	(* Valuto se gli assi sono in finestra di prelievo, in questo modo valuto nel ciclo se devo andare fuori ingombro oppure posso partire da dove sono *)
	//IF Mission^.TPick = TPICK_PACK THEN
	(*	(* Valuto la posizione di X *)
		IF (ModuleAx_X^.Ax^.AxRef^.NcToPlc.SetPos >= WorkPickPoint^[Mission^.PPick].Xv - 50) AND (ModuleAx_X^.Ax^.AxRef^.NcToPlc.SetPos <= WorkPickPoint^[Mission^.PPick].Xv + 50) THEN
			AsseXInFinestraDiPrelievoPacco := TRUE;
		ELSE
			AsseXInFinestraDiPrelievoPacco := FALSE;
		END_IF
		
		(* Valuto la rotazione della pinza *)
		IF ModuleAx_J^.Ax^.AxRef^.NcToPlc.SetPos >= Mission^.JPick - 5 AND ModuleAx_J^.Ax^.AxRef^.NcToPlc.SetPos <= Mission^.JPick + 5 THEN
			AsseJInFinestraDiPrelievoPacco := TRUE;
		ELSE
			AsseJInFinestraDiPrelievoPacco := FALSE;
		END_IF
		
		IF Mission^.JPickVO = 0 THEN //Prelievo Verticale
			IF (ModuleAx_Y^.Ax^.AxRef^.NcToPlc.SetPos  >= WorkPickPoint^[Mission^.PPick].Yv - Mission^.YDim/2 - 50) AND (ModuleAx_Y^.Ax^.AxRef^.NcToPlc.SetPos <= WorkPickPoint^[Mission^.PPick].Yv + Mission^.YDim/2 + 50) THEN
				AsseYInFinestraDiPrelievoPacco := TRUE;
			ELSE
				AsseYInFinestraDiPrelievoPacco := FALSE;
			END_IF
		ELSIF Mission^.JPickVO = 1 THEN//Prelievo Orrizontale
			IF (ModuleAx_Y^.Ax^.AxRef^.NcToPlc.SetPos >= WorkPickPoint^[Mission^.PPick].Yh - Mission^.YDim/2 - 50) AND (ModuleAx_Y^.Ax^.AxRef^.NcToPlc.SetPos <= WorkPickPoint^[Mission^.PPick].Yh + Mission^.YDim/2 + 50) THEN
				AsseYInFinestraDiPrelievoPacco := TRUE;
			ELSE
				AsseYInFinestraDiPrelievoPacco := FALSE;
			END_IF
		END_IF
	
	//END_IF
*)

CASE WorkAreaManager^.State OF
	WAMANAGER_NOP,
	
	WAMANAGER_CICLO_RIPOSO_INIT,
		
	WAMANAGER_CICLO_RIPOSO_RUN:
		IF AbilitaAnticipoDinamico THEN
			QuotaAnticipoDinamicaZ_VersoRiposo := 0;
			
			IF TFDirezioneAssePositiva(Posizione_Attuale:=ModuleAX_X^.Ax^.Status.ActPosition,Posizione_Finale:=Mission^.XPick) THEN	// Direzione Positiva 
				TFCalcolaNumeroPostazioneDXSX(PosizioneAttuale:=ModuleAX_X^.Ax^.Status.ActPosition,
												WorkArea:=WorkArea,
												DirezioneAsseX_Positiva:=TRUE,
												NPostazioneDX=>WADX,
												NPostazioneSX=>WASX,
												PostazionePartenza=>WAPARTENZA);
												
				IF WorkArea^[wa].Typology <> TYPOLOGY_EXTERNAL_DEPPREL THEN
					FOR wa := WAPARTENZA TO NumPostazioneDiPareggiatura DO
						AltezzaDiIngombroArea := 0;
						CASE WorkArea^[wa].Typology OF
							
							TYPOLOGY_PALLET:
								CASE Forming^[WorkAreaState^[wa].F].Pallet.Tipologia OF
										
									PALLET_STANDARD:
										IF WorkAreaState^[wa].H > WorkAreaState^[wa].HPL THEN
											AltezzaDiIngombroArea := WorkAreaState^[wa].H;
										ELSE
											AltezzaDiIngombroArea := WorkAreaState^[wa].HPL;
										END_IF
										IF WorkArea^[wa].Z > AltezzaDiIngombroArea THEN
											AltezzaDiIngombroArea := WorkArea^[wa].Z;	
										END_IF
										
									PALLET_ACCOPPIATI:
										IF WorkAreaState^[wa].H > WorkAreaState^[wa].HPL THEN
											AltezzaDiIngombroArea := WorkAreaState^[wa].H;
										ELSE
											AltezzaDiIngombroArea := WorkAreaState^[wa].HPL;
										END_IF
										IF WorkArea^[wa].Z > AltezzaDiIngombroArea THEN
											AltezzaDiIngombroArea := WorkArea^[wa].Z;	
										END_IF	
									
									CASSA_STANDARD:
										IF Forming^[WorkAreaState^[wa].F].Pallet.HMAX > WorkAreaState^[wa].H THEN
											AltezzaDiIngombroArea := Forming^[WorkAreaState^[wa].F].Pallet.HMAX;
										ELSE
											AltezzaDiIngombroArea := WorkAreaState^[wa].H;
										END_IF
										IF WorkArea^[wa].Z > AltezzaDiIngombroArea THEN
											AltezzaDiIngombroArea := WorkArea^[wa].Z;	
										END_IF
										
									CAVALLETTO:
										IF Forming^[WorkAreaState^[wa].F].Pallet.HMAX > WorkAreaState^[wa].H THEN
											AltezzaDiIngombroArea := Forming^[WorkAreaState^[wa].F].Pallet.HMAX;
										ELSE
											AltezzaDiIngombroArea := WorkAreaState^[wa].H;
										END_IF
										IF WorkArea^[wa].Z > AltezzaDiIngombroArea THEN
											AltezzaDiIngombroArea := WorkArea^[wa].Z;	
										END_IF
										
									BUNDLE:
										IF Forming^[WorkAreaState^[wa].F].Pallet.HMAX > WorkAreaState^[wa].H THEN
											AltezzaDiIngombroArea := Forming^[WorkAreaState^[wa].F].Pallet.HMAX;
										ELSE
											AltezzaDiIngombroArea := WorkAreaState^[wa].H;
										END_IF
										IF WorkArea^[wa].Z > AltezzaDiIngombroArea THEN
											AltezzaDiIngombroArea := WorkArea^[wa].Z;	
										END_IF
										
									ELSE
										AltezzaDiIngombroArea := 1700;//Fisso l'altezza ad una quota di default
								END_CASE
											
							TYPOLOGY_LAYER:
								IF WorkAreaState^[wa].H > WorkAreaState^[wa].HPL THEN
									AltezzaDiIngombroArea := WorkAreaState^[wa].H;
								ELSE
									AltezzaDiIngombroArea := WorkAreaState^[wa].HPL;
								END_IF
								IF WorkArea^[wa].Z > AltezzaDiIngombroArea THEN
									AltezzaDiIngombroArea := WorkArea^[wa].Z;	
								END_IF
							
							TYPOLOGY_EXTERNAL_DEPPREL:
								AltezzaDiIngombroArea := AltezzaDiIngombroArea;
								
							ELSE
								AltezzaDiIngombroArea := 1700;//Fisso l'altezza ad una quota di default
						
						END_CASE					
																
						IF QuotaAnticipoDinamicaZ_VersoRiposo <= AltezzaDiIngombroArea + IngombroZ + OffsetSicurezzaAnticipoMovimenti.OffsetSicurezzaAnticipo_Z THEN
							QuotaAnticipoDinamicaZ_VersoRiposo := AltezzaDiIngombroArea + IngombroZ + OffsetSicurezzaAnticipoMovimenti.OffsetSicurezzaAnticipo_Z;
						END_IF
					END_FOR	
					
				END_IF	
				(* Valuto I Pick-Point *)
				CASE TIPOLOGIA_FUNZIONAMENTO_MACCHINA OF
					
					FUNZIONAMENTO_PICKING:
						AltezzaDiIngombroPuntiPrelievo := 0;
															
				ELSE
					FOR P:=1 TO MAXPICKPOINT DO
						AltezzaDiIngombroPuntiPrelievo := 0;
						IF  WorkPickPointDimension^[P].Zdim + WorkPickPointState^[P].Element.Z >= WorkPickPointDimension^[P].Zdim THEN // Se Altezza + Zpacco >= Ingombro Verticale 
							AltezzaDiIngombroPuntiPrelievo := WorkPickPoint^[P].Z + WorkPickPointState^[P].Element.Z;
						END_IF
						IF WorkPickPointDimension^[P].Zdim >= AltezzaDiIngombroPuntiPrelievo THEN //Se Ingombro Verticale >= Dell'ingombro valutato sopra
							AltezzaDiIngombroPuntiPrelievo := WorkPickPointDimension^[P].Zdim;
						END_IF
						//Se non sono nella WA 7, do una quota fittizzia, inferiore all'altezza del ribaltino "reale"
						IF QuotaAnticipoDinamicaZ_VersoRiposo <= AltezzaDiIngombroPuntiPrelievo + TCPParameter.Z + OffsetSicurezzaAnticipoMovimenti.OffsetSicurezzaAnticipo_Z - 300 THEN
							QuotaAnticipoDinamicaZ_VersoRiposo := AltezzaDiIngombroPuntiPrelievo + WorkPickPointState^[P].Element.YDim + TCPParameter.Z + OffsetSicurezzaAnticipoMovimenti.OffsetSicurezzaAnticipo_Z - 300;
						END_IF
					END_FOR			
				END_CASE
				
			ELSE		// Direzione Negativa
				TFCalcolaNumeroPostazioneDXSX(PosizioneAttuale	:= ModuleAX_X^.Ax^.Status.ActPosition,
												WorkArea		:= WorkArea,
												DirezioneAsseX_Positiva:=FALSE,
												NPostazioneDX	=> WADX,
												NPostazioneSX	=> WASX,
												PostazionePartenza=>WAPARTENZA);
						
				FOR wa := WAPARTENZA TO NPOSTAZIONE_DOPODELPUNTODIPREL BY -1 DO
					AltezzaDiIngombroArea := 0;
					IF WorkAreaState^[wa].H > WorkAreaState^[wa].HPL THEN
						AltezzaDiIngombroArea := WorkAreaState^[wa].H;
					ELSE
						AltezzaDiIngombroArea := WorkAreaState^[wa].HPL;
					END_IF
					IF QuotaAnticipoDinamicaZ_VersoRiposo <= AltezzaDiIngombroArea + TCPParameter.Z + OffsetSicurezzaAnticipoMovimenti.OffsetSicurezzaAnticipo_Z THEN
						QuotaAnticipoDinamicaZ_VersoRiposo := AltezzaDiIngombroArea + TCPParameter.Z + OffsetSicurezzaAnticipoMovimenti.OffsetSicurezzaAnticipo_Z;
					END_IF
				END_FOR			
				(* Valuto I Pick-Point *)
				(*FOR P:=1 TO MAXPICKPOINT DO
					AltezzaDiIngombroPuntiPrelievo := 0;
					IF  WorkPickPoint^[P].Zh + WorkPickPointState^[P].ZDim >= WorkPickPointDimension[P].Zdim THEN // Se Altezza orrizzontale Ribaltino + Zpacco >= Ingombro Verticale Ribaltino
						AltezzaDiIngombroPuntiPrelievo := WorkPickPoint^[P].Zh + WorkPickPointState^[P].ZDim;
					END_IF
					IF WorkPickPoint^[P].Zv + WorkPickPointState^[P].ZTilter + WorkPickPointState^[P].YDim >= WorkPickPointDimension[P].Zdim THEN // Se Altezza Vertivale Ribaltino + Quota Fermo + Ypacco >= Ingombro Verticale Ribaltino
						AltezzaDiIngombroPuntiPrelievo := WorkPickPoint^[P].Zv + WorkPickPointState^[P].ZTilter + WorkPickPointState^[P].YDim;
					END_IF
					IF WorkPickPointDimension[P].Zdim >= AltezzaDiIngombroPuntiPrelievo THEN //Se Ingombro Verticale Ribaltino >= Dell'ingombro valutato sopra
						AltezzaDiIngombroPuntiPrelievo := WorkPickPointDimension[P].Zdim;
					END_IF
					IF WAPARTENZA = NPOSTAZIONE_PRIMADELPUNTODIPREL THEN //Se sono nella posizione 7 valuto l'altezza del ribaltino "REALE", con o senza pacco
						IF QuotaAnticipoDinamicaZ_VersoRiposo <= AltezzaDiIngombroPuntiPrelievo + TCPParameter.Z + OffsetSicurezza.Avuoto THEN //Se Quota fuori ingombro <= dell' ingombro del punto di prelievo
							QuotaAnticipoDinamicaZ_VersoRiposo := AltezzaDiIngombroPuntiPrelievo + TCPParameter.Z + OffsetSicurezza.Avuoto;
						END_IF
					ELSE		//Se non sono nella WA 7, do una quota fittizzia, inferiore all'altezza del ribaltino "reale"
						IF QuotaAnticipoDinamicaZ_VersoRiposo <= AltezzaDiIngombroPuntiPrelievo + TCPParameter.Z + OffsetSicurezzaAnticipoMovimenti.OffsetSicurezzaAnticipo_Z - 300 THEN
							QuotaAnticipoDinamicaZ_VersoRiposo := AltezzaDiIngombroPuntiPrelievo + WorkPickPointState^[P].YDim + TCPParameter.Z + OffsetSicurezzaAnticipoMovimenti.OffsetSicurezzaAnticipo_Z - 300;
						END_IF
					END_IF
				END_FOR*)
			END_IF
			IF ModuleAX_Z^.Ax^.Status.ActPosition >= QuotaAnticipoDinamicaZ_VersoRiposo THEN
				QuotaAnticipoDinamicaZ_Raggiunta := TRUE;
			ELSE
				QuotaAnticipoDinamicaZ_Raggiunta := FALSE;
			END_IF
		END_IF
					
										
	WAMANAGER_CICLO_RIPOSO_END,
			
	(*WAMANAGER_CICLO_PALL_INIT,
	
	WAMANAGER_CICLO_PRELIEVO_PALL_RUN:
		(* Calcolo le WA a DX e a SX della mia posizione attuale *)
		WAPARTENZA := Mission^.PPick;
		TFCalcolaNumeroPostazioneDXSX(PosizioneAttuale	:= ModuleAX_X^.Ax^.Status.ActPosition,
										WorkArea		:= WorkArea,
										NPostazioneDX	=> WADX,
										NPostazioneSX	=> WASX);
																
	WAMANAGER_CICLO_PRELIEVO_PALL_END,						
		
	WAMANAGER_CICLO_DEPOSITO_PALL_RUN:
		IF AbilitaAnticipoDinamico THEN
			QuotaAnticipoDinamicaX_DepositoPallet := 0;	
			QuotaAnticipoDinamicaZ_VersoDepPallet := 0;
						
			//IF DirezioneXPositiva_Dep THEN	// Direzione Positiva 
			IF NOT TFDirezioneAssePositiva(Posizione_Attuale:=ModuleAX_X^.Ax^.Status.ActPosition,Posizione_Finale:=Mission^.XPlace) THEN	// Direzione NEGATIVA 
				FOR wa := WAPARTENZA TO Mission^.PPlace BY -1 DO //ordinamento piazzole CRESCENTE CON LA X
					AltezzaDiIngombroArea := 0;
					IF WorkAreaState^[wa].H > WorkAreaState^[wa].HPL THEN
						AltezzaDiIngombroArea := WorkAreaState^[wa].H;
					ELSE
						AltezzaDiIngombroArea := WorkAreaState^[wa].HPL;
					END_IF
					IF QuotaAnticipoDinamicaZ_VersoDepPallet <= AltezzaDiIngombroArea + TCPParameter.Z + OffsetSicurezzaAnticipoMovimenti.OffsetSicurezzaAnticipo_Z THEN
						QuotaAnticipoDinamicaZ_VersoDepPallet := AltezzaDiIngombroArea + TCPParameter.Z + OffsetSicurezzaAnticipoMovimenti.OffsetSicurezzaAnticipo_Z;
					END_IF
				END_FOR		
				(* Valuto I Pick-Point *)
				(*FOR P:=1 TO MAXPICKPOINT DO
					AltezzaDiIngombroPuntiPrelievo := 0;
					IF  WorkPickPoint^[P].Zh + WorkPickPointState^[P].ZDim >= WorkPickPointDimension[P].Zdim THEN // Se Altezza orrizzontale Ribaltino + Zpacco >= Ingombro Verticale Ribaltino
						AltezzaDiIngombroPuntiPrelievo := WorkPickPoint^[P].Zh + WorkPickPointState^[P].ZDim;
					END_IF
					IF WorkPickPoint^[P].Zv + WorkPickPointState^[P].ZTilter + WorkPickPointState^[P].YDim >= WorkPickPointDimension[P].Zdim THEN // Se Altezza Vertivale Ribaltino + Quota Fermo + Ypacco >= Ingombro Verticale Ribaltino
						AltezzaDiIngombroPuntiPrelievo := WorkPickPoint^[P].Zv + WorkPickPointState^[P].ZTilter + WorkPickPointState^[P].YDim;
					END_IF
					IF WorkPickPointDimension[P].Zdim >= AltezzaDiIngombroPuntiPrelievo THEN //Se Ingombro Verticale Ribaltino >= Dell'ingombro valutato sopra
						AltezzaDiIngombroPuntiPrelievo := WorkPickPointDimension[P].Zdim;
					END_IF
					IF WAPARTENZA = NPOSTAZIONE_DOPORIBALTINO THEN //ACR:Se sono nella posizione 7 valuto l'altezza del ribaltino "REALE", con o senza pacco
						IF QuotaAnticipoDinamicaZ_VersoDepPallet <= AltezzaDiIngombroPuntiPrelievo + TCPParameter.Z + OffsetSicurezza.Avuoto THEN //Se Quota fuori ingombro <= dell' ingombro del punto di prelievo
							QuotaAnticipoDinamicaZ_VersoDepPallet := AltezzaDiIngombroPuntiPrelievo + TCPParameter.Z + OffsetSicurezza.Avuoto;
						END_IF
					ELSE		//ACR:Se non sono nella WA 7, do una quota fittizzia, inferiore all'altezza del ribaltino "reale"
						IF QuotaAnticipoDinamicaZ_VersoDepPallet <= AltezzaDiIngombroPuntiPrelievo + TCPParameter.Z + OffsetSicurezzaAnticipoMovimenti.OffsetSicurezzaAnticipo_Z - 300 THEN
							QuotaAnticipoDinamicaZ_VersoDepPallet := AltezzaDiIngombroPuntiPrelievo + WorkPickPointState^[P].YDim + TCPParameter.Z + OffsetSicurezzaAnticipoMovimenti.OffsetSicurezzaAnticipo_Z - 300;
						END_IF
					END_IF
				END_FOR*)
			ELSE		// Direzione POSITIVA
				FOR wa := WAPARTENZA TO Mission^.PPlace DO
					AltezzaDiIngombroArea := 0;
					IF WorkAreaState^[wa].H > WorkAreaState^[wa].HPL THEN
						AltezzaDiIngombroArea := WorkAreaState^[wa].H;
					ELSE
						AltezzaDiIngombroArea := WorkAreaState^[wa].HPL;
					END_IF
					IF QuotaAnticipoDinamicaZ_VersoDepPallet <= AltezzaDiIngombroArea + TCPParameter.Z + OffsetSicurezzaAnticipoMovimenti.OffsetSicurezzaAnticipo_Z THEN
						QuotaAnticipoDinamicaZ_VersoDepPallet := AltezzaDiIngombroArea + TCPParameter.Z + OffsetSicurezzaAnticipoMovimenti.OffsetSicurezzaAnticipo_Z;
					END_IF
				END_FOR			
				(* Valuto I Pick-Point *)
				(*FOR P:=1 TO MAXPICKPOINT DO
					AltezzaDiIngombroPuntiPrelievo := 0;
					IF  WorkPickPoint^[P].Zh + WorkPickPointState^[P].ZDim >= WorkPickPointDimension[P].Zdim THEN // Se Altezza orrizzontale Ribaltino + Zpacco >= Ingombro Verticale Ribaltino
						AltezzaDiIngombroPuntiPrelievo := WorkPickPoint^[P].Zh + WorkPickPointState^[P].ZDim;
					END_IF
					IF WorkPickPoint^[P].Zv + WorkPickPointState^[P].ZTilter + WorkPickPointState^[P].YDim >= WorkPickPointDimension[P].Zdim THEN // Se Altezza Vertivale Ribaltino + Quota Fermo + Ypacco >= Ingombro Verticale Ribaltino
						AltezzaDiIngombroPuntiPrelievo := WorkPickPoint^[P].Zv + WorkPickPointState^[P].ZTilter + WorkPickPointState^[P].YDim;
					END_IF
					IF WorkPickPointDimension[P].Zdim >= AltezzaDiIngombroPuntiPrelievo THEN //Se Ingombro Verticale Ribaltino >= Dell'ingombro valutato sopra
						AltezzaDiIngombroPuntiPrelievo := WorkPickPointDimension[P].Zdim;
					END_IF
					IF WAPARTENZA = NPOSTAZIONE_PRIMADELPUNTODIPREL THEN //Se sono nella posizione 7 valuto l'altezza del ribaltino "REALE", con o senza pacco
						IF QuotaAnticipoDinamicaZ_VersoDepPallet <= AltezzaDiIngombroPuntiPrelievo + TCPParameter.Z + OffsetSicurezza.Avuoto THEN //Se Quota fuori ingombro <= dell' ingombro del punto di prelievo
							QuotaAnticipoDinamicaZ_VersoDepPallet := AltezzaDiIngombroPuntiPrelievo + TCPParameter.Z + OffsetSicurezza.Avuoto;
						END_IF
					ELSE		//Se non sono nella WA 7, do una quota fittizzia, inferiore all'altezza del ribaltino "reale"
						IF QuotaAnticipoDinamicaZ_VersoDepPallet <= AltezzaDiIngombroPuntiPrelievo + TCPParameter.Z + OffsetSicurezzaAnticipoMovimenti.OffsetSicurezzaAnticipo_Z - 300 THEN
							QuotaAnticipoDinamicaZ_VersoDepPallet := AltezzaDiIngombroPuntiPrelievo + WorkPickPointState^[P].YDim + TCPParameter.Z + OffsetSicurezzaAnticipoMovimenti.OffsetSicurezzaAnticipo_Z - 300;
						END_IF
					END_IF
				END_FOR*)
				IF ModuleAX_Z^.Ax^.Status.ActPosition >= QuotaAnticipoDinamicaZ_VersoDepPallet THEN
					QuotaAnticipoDinamicaZ_Raggiunta := TRUE;
				ELSE
					QuotaAnticipoDinamicaZ_Raggiunta := FALSE;
				END_IF	
			END_IF
					
		////////////////// ANTICIPO X ///////////////////////
	(*	IF TFDirezioneAssePositiva(Posizione_Attuale:=ModuleAX_X^.Ax^.Status.ActPosition,Posizione_Finale:=Mission^.XPlace) THEN // Direzione Positiva
			IF Mission^.PPlace <= NPOSTAZIONE_PRIMADELPUNTODIPREL THEN
				IF WorkAreaState^[Mission^.PPlace + 1].P <= 1 THEN
					QuotaAnticipoDinamicaX_DepositoPallet := (Workarea^[Mission^.PPlace + 1].X - Pallet^[Workarea^[Mission^.PPlace + 1].Pallet].X/2 + OffsetSicurezzaAnticipoMovimenti.OffsetSicurezzaAnticipo_X + (IngombroX/2));
				ELSE
					QuotaAnticipoDinamicaX_DepositoPallet := (Workarea^[Mission^.PPlace + 1].X + Pallet^[Workarea^[Mission^.PPlace + 1].Pallet].X/2 + OffsetSicurezzaAnticipoMovimenti.OffsetSicurezzaAnticipo_X + (IngombroX/2));
				END_IF	
			ELSIF Mission^.PPlace > NPOSTAZIONE_DOPORIBALTINO THEN
				IF WorkAreaState^[Mission^.PPlace + 1].P <= 1 THEN
					QuotaAnticipoDinamicaX_DepositoPallet := (Workarea^[Mission^.PPlace + 1].X - Pallet^[Workarea^[Mission^.PPlace + 1].Pallet].X/2 + OffsetSicurezzaAnticipoMovimenti.OffsetSicurezzaAnticipo_X + (IngombroX/2));
				ELSE
					QuotaAnticipoDinamicaX_DepositoPallet := (Workarea^[Mission^.PPlace + 1].X + Pallet^[Workarea^[Mission^.PPlace + 1].Pallet].X/2 + OffsetSicurezzaAnticipoMovimenti.OffsetSicurezzaAnticipo_X + (IngombroX/2));
				END_IF
				IF QuotaAnticipoDinamicaX_DepositoPallet <= Workarea^[NPOSTAZIONE_DOPORIBALTINO].X (*+ 800*) THEN // +800 : In ACR la wa 6 è occupata da falde, questo valore ne indica l'ingombro dal centro verso la wa n° 5
					QuotaAnticipoDinamicaX_DepositoPallet := Workarea^[NPOSTAZIONE_DOPORIBALTINO].X (*+ 800*);
				END_IF
			ELSIF Mission^.PPlace = NPOSTAZIONE_DOPORIBALTINO THEN //postazione 6
				QuotaAnticipoDinamicaX_DepositoPallet := (WorkPickPoint^[Mission^.PPick].Xv + LarghezzaPickPoint/2 + OffsetSicurezzaAnticipoMovimenti.OffsetSicurezzaAnticipo_X + (IngombroX/2));
			END_IF
			IF ModuleAX_X^.Ax^.Status.ActPosition >= QuotaAnticipoDinamicaX_DepositoPallet THEN
				QuotaAnticipoDinamicaX_Raggiunta := TRUE;
			ELSE
				QuotaAnticipoDinamicaX_Raggiunta := FALSE;
			END_IF
		ELSE	//Direzione Negativa
			IF Mission^.PPlace < NPOSTAZIONE_PRIMADELPUNTODIPREL OR Mission^.PPlace >= NPOSTAZIONE_DOPORIBALTINO THEN
				IF WorkAreaState^[Mission^.PPlace - 1].P <= 1 THEN
					QuotaAnticipoDinamicaX_DepositoPallet := (Workarea^[Mission^.PPlace - 1].X + Pallet^[Workarea^[Mission^.PPlace - 1].Pallet].X/2 - OffsetSicurezzaAnticipoMovimenti.OffsetSicurezzaAnticipo_X - (IngombroX/2));
				ELSE
					QuotaAnticipoDinamicaX_DepositoPallet := (Workarea^[Mission^.PPlace - 1].X - Pallet^[Workarea^[Mission^.PPlace - 1].Pallet].X/2 - OffsetSicurezzaAnticipoMovimenti.OffsetSicurezzaAnticipo_X - (IngombroX/2));
				END_IF
			ELSIF Mission^.PPlace = NPOSTAZIONE_PRIMADELPUNTODIPREL THEN
				QuotaAnticipoDinamicaX_DepositoPallet := (WorkPickPoint^[Mission^.PPick].Xv - LarghezzaPickPoint/2 - OffsetSicurezzaAnticipoMovimenti.OffsetSicurezzaAnticipo_X - (IngombroX/2));
			END_IF
			IF ModuleAX_X^.Ax^.Status.ActPosition <= QuotaAnticipoDinamicaX_DepositoPallet THEN
				QuotaAnticipoDinamicaX_Raggiunta := TRUE;
			ELSE
				QuotaAnticipoDinamicaX_Raggiunta := FALSE;
			END_IF
		END_IF*)
		
	END_IF	
				
	WAMANAGER_CICLO_DEPOSITO_PALL_END,
	
	WAMANAGER_CICLO_FALDA_VUOTI_INIT,
	
	WAMANAGER_CICLO_PRELIEVO_FALDA_VUOTI_RUN:
		IF AbilitaAnticipoDinamico THEN
			QuotaAnticipoDinamicaZ_VersoPrelFalda := 0;
				
			//IF DirezioneXPositiva_Prel THEN	// Direzione Positiva 
			IF NOT TFDirezioneAssePositiva(Posizione_Attuale:=ModuleAX_X^.Ax^.Status.ActPosition,Posizione_Finale:=Mission^.XPick) THEN	// Direzione NEGATIVA 
				TFCalcolaNumeroPostazioneDXSX(PosizioneAttuale	:= ModuleAX_X^.Ax^.Status.ActPosition,
												WorkArea		:= WorkArea,
												DirezioneAsseX_Positiva := FALSE,
												NPostazioneDX	=> WADX,
												NPostazioneSX	=> WASX,
												PostazionePartenza=>WAPARTENZA);
				
				FOR wa := WAPARTENZA TO 1 BY -1 DO
					AltezzaDiIngombroArea := 0;
					IF WorkAreaState^[wa].H > WorkAreaState^[wa].HPL THEN
						AltezzaDiIngombroArea := WorkAreaState^[wa].H;
					ELSE
						AltezzaDiIngombroArea := WorkAreaState^[wa].HPL;
					END_IF
					IF QuotaAnticipoDinamicaZ_VersoPrelFalda <= AltezzaDiIngombroArea + TCPParameter.Z + OffsetSicurezzaAnticipoMovimenti.OffsetSicurezzaAnticipo_Z THEN
						QuotaAnticipoDinamicaZ_VersoPrelFalda := AltezzaDiIngombroArea + TCPParameter.Z + OffsetSicurezzaAnticipoMovimenti.OffsetSicurezzaAnticipo_Z;
					END_IF
				END_FOR		
				
				(* Valuto I Pick-Point *)
				(*FOR P:=1 TO MAXPICKPOINT DO
					AltezzaDiIngombroPuntiPrelievo := 0;
					IF  WorkPickPoint^[P].Zh + WorkPickPointState^[P].ZDim >= WorkPickPointDimension[P].Zdim THEN // Se Altezza orrizzontale Ribaltino + Zpacco >= Ingombro Verticale Ribaltino
						AltezzaDiIngombroPuntiPrelievo := WorkPickPoint^[P].Zh + WorkPickPointState^[P].ZDim;
					END_IF
					IF WorkPickPoint^[P].Zv + WorkPickPointState^[P].ZTilter + WorkPickPointState^[P].YDim >= WorkPickPointDimension[P].Zdim THEN // Se Altezza Vertivale Ribaltino + Quota Fermo + Ypacco >= Ingombro Verticale Ribaltino
						AltezzaDiIngombroPuntiPrelievo := WorkPickPoint^[P].Zv + WorkPickPointState^[P].ZTilter + WorkPickPointState^[P].YDim;
					END_IF
					IF WorkPickPointDimension[P].Zdim >= AltezzaDiIngombroPuntiPrelievo THEN //Se Ingombro Verticale Ribaltino >= Dell'ingombro valutato sopra
						AltezzaDiIngombroPuntiPrelievo := WorkPickPointDimension[P].Zdim;
					END_IF
					IF QuotaAnticipoDinamicaZ_VersoPrelFalda <= AltezzaDiIngombroPuntiPrelievo + TCPParameter.Z + OffsetSicurezza.Avuoto THEN //Se Quota fuori ingombro <= dell' ingombro del punto di prelievo
						QuotaAnticipoDinamicaZ_VersoPrelFalda := AltezzaDiIngombroPuntiPrelievo + TCPParameter.Z + OffsetSicurezza.Avuoto;
					END_IF	
				END_FOR*)
				
			ELSE		// Direzione POSITIVA
				FOR wa := WAPARTENZA TO MAXAREA DO
					AltezzaDiIngombroArea := 0;
					IF WorkAreaState^[wa].H > WorkAreaState^[wa].HPL THEN
						AltezzaDiIngombroArea := WorkAreaState^[wa].H;
					ELSE
						AltezzaDiIngombroArea := WorkAreaState^[wa].HPL;
					END_IF
					IF QuotaAnticipoDinamicaZ_VersoPrelFalda <= AltezzaDiIngombroArea + TCPParameter.Z + OffsetSicurezzaAnticipoMovimenti.OffsetSicurezzaAnticipo_Z THEN
						QuotaAnticipoDinamicaZ_VersoPrelFalda := AltezzaDiIngombroArea + TCPParameter.Z + OffsetSicurezzaAnticipoMovimenti.OffsetSicurezzaAnticipo_Z;
					END_IF
				END_FOR			
				(* Valuto I Pick-Point *)
				(*FOR P:=1 TO MAXPICKPOINT DO
					IF Mission^.JPickVO = 0 THEN //Ribaltino Verticale
						IF QuotaAnticipoDinamicaZ_VersoPrelFalda <= WorkPickPoint^[P].Zv + WorkPickPointState^[P].ZTilter + WorkPickPointState^[P].YDim + TCPParameter.Z + OffsetSicurezzaAnticipoMovimenti.OffsetSicurezzaAnticipo_Z THEN
							QuotaAnticipoDinamicaZ_VersoPrelFalda := WorkPickPoint^[P].Zv + WorkPickPointState^[P].ZTilter + WorkPickPointState^[P].YDim + TCPParameter.Z + OffsetSicurezzaAnticipoMovimenti.OffsetSicurezzaAnticipo_Z;
						END_IF
					ELSIF Mission^.JPickVO = 1 THEN	//Ribaltino Orrizontale
						IF QuotaAnticipoDinamicaZ_VersoPrelFalda <= WorkPickPoint^[P].Zh + WorkPickPointState^[P].ZDim + TCPParameter.Z + OffsetSicurezzaAnticipoMovimenti.OffsetSicurezzaAnticipo_Z THEN
							QuotaAnticipoDinamicaZ_VersoPrelFalda := WorkPickPoint^[P].Zh + WorkPickPointState^[P].ZDim + TCPParameter.Z + OffsetSicurezzaAnticipoMovimenti.OffsetSicurezzaAnticipo_Z;
						END_IF
					ELSE
						QuotaAnticipoDinamicaZ_VersoPrelFalda := ALTEZZA_CATASTA_FALDE; // Misura di sicurezza fittizzia
					END_IF
				END_FOR*)
			END_IF
			IF ModuleAX_Z^.Ax^.Status.ActPosition >= QuotaAnticipoDinamicaZ_VersoPrelFalda THEN
				QuotaAnticipoDinamicaZ_Raggiunta := TRUE;
			ELSE
				QuotaAnticipoDinamicaZ_Raggiunta := FALSE;
			END_IF
		END_IF
		
						
	WAMANAGER_CICLO_PRELIEVO_FALDA_VUOTI_END,
		
	WAMANAGER_CICLO_DEPOSITO_FALDA_VUOTI_RUN:
		IF AbilitaAnticipoDinamico THEN
			QuotaAnticipoDinamicaX_VersoDepFalda := 0;
			
			IF TFDirezioneAssePositiva(Posizione_Attuale:=ModuleAX_X^.Ax^.Status.ActPosition,Posizione_Finale:=Mission^.XPlace) THEN
															
				(*IF Mission^.PPlace <= NPOSTAZIONE_PRIMADELPUNTODIPREL THEN
					IF WorkAreaState^[Mission^.PPlace + 1].P <= 1 THEN
						QuotaAnticipoDinamicaX_VersoDepFalda := (Workarea^[Mission^.PPlace + 1].X - Pallet^[Workarea^[Mission^.PPlace + 1].Pallet].X/2 + OffsetSicurezzaAnticipoMovimenti.OffsetSicurezzaAnticipo_X + (IngombroX/2));
					ELSE
						QuotaAnticipoDinamicaX_VersoDepFalda := (Workarea^[Mission^.PPlace + 1].X + Pallet^[Workarea^[Mission^.PPlace + 1].Pallet].X/2 + OffsetSicurezzaAnticipoMovimenti.OffsetSicurezzaAnticipo_X + (IngombroX/2));
					END_IF	
				ELSIF Mission^.PPlace > NPOSTAZIONE_DOPORIBALTINO THEN
					IF WorkAreaState^[Mission^.PPlace + 1].P <= 1 THEN
						QuotaAnticipoDinamicaX_VersoDepFalda := (Workarea^[Mission^.PPlace + 1].X - Pallet^[Workarea^[Mission^.PPlace + 1].Pallet].X/2 + OffsetSicurezzaAnticipoMovimenti.OffsetSicurezzaAnticipo_X + (IngombroX/2));
					ELSE
						QuotaAnticipoDinamicaX_VersoDepFalda := (Workarea^[Mission^.PPlace + 1].X + Pallet^[Workarea^[Mission^.PPlace + 1].Pallet].X/2 + OffsetSicurezzaAnticipoMovimenti.OffsetSicurezzaAnticipo_X + (IngombroX/2));
					END_IF
					IF QuotaAnticipoDinamicaX_VersoDepFalda <= Workarea^[NPOSTAZIONE_DOPORIBALTINO].X + 800 THEN
						QuotaAnticipoDinamicaX_VersoDepFalda := Workarea^[NPOSTAZIONE_DOPORIBALTINO].X + 800;
					END_IF
				ELSIF Mission^.PPlace = NPOSTAZIONE_DOPORIBALTINO THEN //postazione 6
					QuotaAnticipoDinamicaX_VersoDepFalda := (WorkPickPoint^[Mission^.PPick].Xv + LarghezzaPickPoint/2 + OffsetSicurezzaAnticipoMovimenti.OffsetSicurezzaAnticipo_X + (IngombroX/2));
				END_IF
				IF ModuleAX_X^.Ax^.Status.ActPosition >= QuotaAnticipoDinamicaX_VersoDepFalda THEN
					QuotaAnticipoDinamicaX_Raggiunta := TRUE;
				ELSE
					QuotaAnticipoDinamicaX_Raggiunta := FALSE;
				END_IF
			ELSE	//Direzione Negativa
				IF Mission^.PPlace < NPOSTAZIONE_PRIMADELPUNTODIPREL OR Mission^.PPlace >= NPOSTAZIONE_DOPORIBALTINO THEN
					IF WorkAreaState^[Mission^.PPlace - 1].P <= 1 OR WorkArea^[Mission^.PPlace - 1].H + 100 < WorkArea^[Mission^.PPlace].H  THEN
						QuotaAnticipoDinamicaX_VersoDepFalda := (Workarea^[Mission^.PPlace - 1].X + Pallet^[Workarea^[Mission^.PPlace - 1].Pallet].X/2 - OffsetSicurezzaAnticipoMovimenti.OffsetSicurezzaAnticipo_X - (IngombroX/2));
					ELSE
						QuotaAnticipoDinamicaX_VersoDepFalda := (Workarea^[Mission^.PPlace - 1].X - Pallet^[Workarea^[Mission^.PPlace - 1].Pallet].X/2 - OffsetSicurezzaAnticipoMovimenti.OffsetSicurezzaAnticipo_X - (IngombroX/2));
					END_IF
				ELSIF Mission^.PPlace = NPOSTAZIONE_PRIMADELPUNTODIPREL THEN
					QuotaAnticipoDinamicaX_VersoDepFalda := (WorkPickPoint^[Mission^.PPick].Xv - LarghezzaPickPoint/2 - OffsetSicurezzaAnticipoMovimenti.OffsetSicurezzaAnticipo_X - (IngombroX/2));
				END_IF
				IF ModuleAX_X^.Ax^.Status.ActPosition <= QuotaAnticipoDinamicaX_VersoDepFalda THEN
					QuotaAnticipoDinamicaX_Raggiunta := TRUE;
				ELSE
					QuotaAnticipoDinamicaX_Raggiunta := FALSE;
				END_IF*);
			END_IF
		END_IF
											
	WAMANAGER_CICLO_DEPOSITO_FALDA_VUOTI_END,*)
	
	WAMANAGER_CICLO_FALDA_INIT,
	
	WAMANAGER_CICLO_PRELIEVO_FALDA_RUN:
		QuotaAnticipoDinamicaX_Raggiunta := FALSE;
		QuotaAnticipoDinamicaZ_Raggiunta := FALSE;
		QuotaAnticipoDinamicaZ_VersoPrelFalda := 0;
		IF AbilitaAnticipoDinamico THEN
			
			//IF DirezioneXPositiva_Prel THEN	// Direzione Positiva 
			IF NOT TFDirezioneAssePositiva(Posizione_Attuale:=ModuleAX_X^.Ax^.Status.ActPosition,Posizione_Finale:=Mission^.XPlace) THEN	// Direzione NEGATIVA 
				FOR wa := WAPARTENZA TO 1 BY -1 DO
					AltezzaDiIngombroArea := 0;
					IF WorkAreaState^[wa].H > WorkAreaState^[wa].HPL THEN
						AltezzaDiIngombroArea := WorkAreaState^[wa].H;
					ELSE
						AltezzaDiIngombroArea := WorkAreaState^[wa].HPL;
					END_IF
					IF QuotaAnticipoDinamicaZ_VersoPrelFalda <= AltezzaDiIngombroArea + TCPParameter.Z + OffsetSicurezzaAnticipoMovimenti.OffsetSicurezzaAnticipo_Z THEN
						QuotaAnticipoDinamicaZ_VersoPrelFalda := AltezzaDiIngombroArea + TCPParameter.Z + OffsetSicurezzaAnticipoMovimenti.OffsetSicurezzaAnticipo_Z;
					END_IF
				END_FOR		
				
				(* Valuto I Pick-Point *)
				(*FOR P:=1 TO MAXPICKPOINT DO
					AltezzaDiIngombroPuntiPrelievo := 0;
					IF  WorkPickPoint^[P].Zh + WorkPickPointState^[P].ZDim >= WorkPickPointDimension[P].Zdim THEN // Se Altezza orrizzontale Ribaltino + Zpacco >= Ingombro Verticale Ribaltino
						AltezzaDiIngombroPuntiPrelievo := WorkPickPoint^[P].Zh + WorkPickPointState^[P].ZDim;
					END_IF
					IF WorkPickPoint^[P].Zv + WorkPickPointState^[P].ZTilter + WorkPickPointState^[P].YDim >= WorkPickPointDimension[P].Zdim THEN // Se Altezza Vertivale Ribaltino + Quota Fermo + Ypacco >= Ingombro Verticale Ribaltino
						AltezzaDiIngombroPuntiPrelievo := WorkPickPoint^[P].Zv + WorkPickPointState^[P].ZTilter + WorkPickPointState^[P].YDim;
					END_IF
					IF WorkPickPointDimension[P].Zdim >= AltezzaDiIngombroPuntiPrelievo THEN //Se Ingombro Verticale Ribaltino >= Dell'ingombro valutato sopra
						AltezzaDiIngombroPuntiPrelievo := WorkPickPointDimension[P].Zdim;
					END_IF
					IF QuotaAnticipoDinamicaZ_VersoPrelFalda <= AltezzaDiIngombroPuntiPrelievo + TCPParameter.Z + OffsetSicurezza.Avuoto THEN //Se Quota fuori ingombro <= dell' ingombro del punto di prelievo
						QuotaAnticipoDinamicaZ_VersoPrelFalda := AltezzaDiIngombroPuntiPrelievo + TCPParameter.Z + OffsetSicurezza.Avuoto;
					END_IF	
				END_FOR*)
				
			ELSE		// Direzione Negativa
				FOR wa := WAPARTENZA TO MAXAREAPRESENT DO
					AltezzaDiIngombroArea := 0;
					IF WorkAreaState^[wa].H > WorkAreaState^[wa].HPL THEN
						AltezzaDiIngombroArea := WorkAreaState^[wa].H;
					ELSE
						AltezzaDiIngombroArea := WorkAreaState^[wa].HPL;
					END_IF
					IF QuotaAnticipoDinamicaZ_VersoPrelFalda <= AltezzaDiIngombroArea + TCPParameter.Z + OffsetSicurezzaAnticipoMovimenti.OffsetSicurezzaAnticipo_Z THEN
						QuotaAnticipoDinamicaZ_VersoPrelFalda := AltezzaDiIngombroArea + TCPParameter.Z + OffsetSicurezzaAnticipoMovimenti.OffsetSicurezzaAnticipo_Z;
					END_IF
				END_FOR			
				(* Valuto I Pick-Point *)
				(*FOR P:=1 TO MAXPICKPOINT DO
					IF Mission^.JPickVO = 0 THEN //Ribaltino Verticale
						IF QuotaAnticipoDinamicaZ_VersoPrelFalda <= WorkPickPoint^[P].Zv + WorkPickPointState^[P].ZTilter + WorkPickPointState^[P].YDim + TCPParameter.Z + OffsetSicurezzaAnticipoMovimenti.OffsetSicurezzaAnticipo_Z THEN
							QuotaAnticipoDinamicaZ_VersoPrelFalda := WorkPickPoint^[P].Zv + WorkPickPointState^[P].ZTilter + WorkPickPointState^[P].YDim + TCPParameter.Z + OffsetSicurezzaAnticipoMovimenti.OffsetSicurezzaAnticipo_Z;
						END_IF
					ELSIF Mission^.JPickVO = 1 THEN	//Ribaltino Orrizontale
						IF QuotaAnticipoDinamicaZ_VersoPrelFalda <= WorkPickPoint^[P].Zh + WorkPickPointState^[P].ZDim + TCPParameter.Z + OffsetSicurezzaAnticipoMovimenti.OffsetSicurezzaAnticipo_Z THEN
							QuotaAnticipoDinamicaZ_VersoPrelFalda := WorkPickPoint^[P].Zh + WorkPickPointState^[P].ZDim + TCPParameter.Z + OffsetSicurezzaAnticipoMovimenti.OffsetSicurezzaAnticipo_Z;
						END_IF
					ELSE
						QuotaAnticipoDinamicaZ_VersoPrelFalda := ALTEZZA_CATASTA_FALDE; // Misura di sicurezza fittizzia
					END_IF
				END_FOR*)
			END_IF
			IF ModuleAX_Z^.Ax^.Status.ActPosition >= QuotaAnticipoDinamicaZ_VersoPrelFalda THEN
				QuotaAnticipoDinamicaZ_Raggiunta := TRUE;
			ELSE
				QuotaAnticipoDinamicaZ_Raggiunta := FALSE;
			END_IF
		END_IF
		
													
	WAMANAGER_CICLO_PRELIEVO_FALDA_END,
			
	WAMANAGER_CICLO_DEPOSITO_FALDA_RUN:
		IF AbilitaAnticipoDinamico THEN
			QuotaAnticipoDinamicaX_VersoDepFalda := 0;
						
			(*IF TFDirezioneAssePositiva(Posizione_Attuale:=ModuleAX_X^.Ax^.Status.ActPosition,Posizione_Finale:=Mission^.XPlace) THEN
				IF Mission^.PPlace <= NPOSTAZIONE_PRIMADELPUNTODIPREL THEN
					IF WorkAreaState^[Mission^.PPlace + 1].P <= 1 THEN
						QuotaAnticipoDinamicaX_VersoDepFalda := (Workarea^[Mission^.PPlace + 1].X - Pallet^[Workarea^[Mission^.PPlace + 1].Pallet].X/2 + OffsetSicurezzaAnticipoMovimenti.OffsetSicurezzaAnticipo_X + (IngombroX/2));
					ELSE
						QuotaAnticipoDinamicaX_VersoDepFalda := (Workarea^[Mission^.PPlace + 1].X + Pallet^[Workarea^[Mission^.PPlace + 1].Pallet].X/2 + OffsetSicurezzaAnticipoMovimenti.OffsetSicurezzaAnticipo_X + (IngombroX/2));
					END_IF	
				ELSIF Mission^.PPlace > NPOSTAZIONE_DOPORIBALTINO THEN
					IF WorkAreaState^[Mission^.PPlace + 1].P <= 1 THEN
						QuotaAnticipoDinamicaX_VersoDepFalda := (Workarea^[Mission^.PPlace + 1].X - Pallet^[Workarea^[Mission^.PPlace + 1].Pallet].X/2 + OffsetSicurezzaAnticipoMovimenti.OffsetSicurezzaAnticipo_X + (IngombroX/2));
					ELSE
						QuotaAnticipoDinamicaX_VersoDepFalda := (Workarea^[Mission^.PPlace + 1].X + Pallet^[Workarea^[Mission^.PPlace + 1].Pallet].X/2 + OffsetSicurezzaAnticipoMovimenti.OffsetSicurezzaAnticipo_X + (IngombroX/2));
					END_IF
					IF QuotaAnticipoDinamicaX_VersoDepFalda <= Workarea^[NPOSTAZIONE_DOPORIBALTINO].X + 800 THEN
						QuotaAnticipoDinamicaX_VersoDepFalda := Workarea^[NPOSTAZIONE_DOPORIBALTINO].X + 800;
					END_IF
				ELSIF Mission^.PPlace = NPOSTAZIONE_DOPORIBALTINO THEN //postazione 6
					QuotaAnticipoDinamicaX_VersoDepFalda := (WorkPickPoint^[Mission^.PPick].Xv + LarghezzaPickPoint/2 + OffsetSicurezzaAnticipoMovimenti.OffsetSicurezzaAnticipo_X + (IngombroX/2));
				END_IF
				IF ModuleAX_X^.Ax^.Status.ActPosition >= QuotaAnticipoDinamicaX_VersoDepFalda THEN
					QuotaAnticipoDinamicaX_Raggiunta := TRUE;
				ELSE
					QuotaAnticipoDinamicaX_Raggiunta := FALSE;
				END_IF
				TFCalcolaNumeroPostazioneDXSX(PosizioneAttuale	:= ModuleAX_X^.Ax^.Status.ActPosition,
												WorkArea		:= WorkArea,
												DirezioneAsseX_Positiva := TRUE,
												NPostazioneDX	=> WADX,
												NPostazioneSX	=> WASX,
												PostazionePartenza=>WAPARTENZA);
			ELSE	//Direzione Negativa
				IF Mission^.PPlace < NPOSTAZIONE_PRIMADELPUNTODIPREL OR Mission^.PPlace >= NPOSTAZIONE_DOPORIBALTINO THEN
					IF WorkAreaState^[Mission^.PPlace - 1].P <= 1 OR WorkArea^[Mission^.PPlace - 1].H + 100 < WorkArea^[Mission^.PPlace].H  THEN
						QuotaAnticipoDinamicaX_VersoDepFalda := (Workarea^[Mission^.PPlace - 1].X + Pallet^[Workarea^[Mission^.PPlace - 1].Pallet].X/2 - OffsetSicurezzaAnticipoMovimenti.OffsetSicurezzaAnticipo_X - (IngombroX/2));
					ELSE
						QuotaAnticipoDinamicaX_VersoDepFalda := (Workarea^[Mission^.PPlace - 1].X - Pallet^[Workarea^[Mission^.PPlace - 1].Pallet].X/2 - OffsetSicurezzaAnticipoMovimenti.OffsetSicurezzaAnticipo_X - (IngombroX/2));
					END_IF
				ELSIF Mission^.PPlace = NPOSTAZIONE_PRIMADELPUNTODIPREL THEN
					QuotaAnticipoDinamicaX_VersoDepFalda := (WorkPickPoint^[Mission^.PPick].Xv - LarghezzaPickPoint/2 - OffsetSicurezzaAnticipoMovimenti.OffsetSicurezzaAnticipo_X - (IngombroX/2));
				END_IF
				IF ModuleAX_X^.Ax^.Status.ActPosition <= QuotaAnticipoDinamicaX_VersoDepFalda THEN
					QuotaAnticipoDinamicaX_Raggiunta := TRUE;
				ELSE
					QuotaAnticipoDinamicaX_Raggiunta := FALSE;
				END_IF
			END_IF
			TFCalcolaNumeroPostazioneDXSX(PosizioneAttuale	:= ModuleAX_X^.Ax^.Status.ActPosition,
												WorkArea		:= WorkArea,
												DirezioneAsseX_Positiva := FALSE,
												NPostazioneDX	=> WADX,
												NPostazioneSX	=> WASX,
												PostazionePartenza=>WAPARTENZA);
			*)
		END_IF
		WAPARTENZA := Mission^.PPlace;
				
	//WAMANAGER_CICLO_DEPOSITO_FALDA_END,

	(*WAMANAGER_CICLO_PACCO_INIT,
	
	WAMANAGER_CICLO_PRELIEVO_PACCO_RUN:
		IF AbilitaAnticipoDinamico THEN
			QuotaAnticipoDinamicaZ_VersoPrelPacco := 0; 
			//IF DirezioneXPositiva_Prel THEN	// Direzione Positiva 
			IF NOT TFDirezioneAssePositiva(Posizione_Attuale:=ModuleAX_X^.Ax^.Status.ActPosition,Posizione_Finale:=Mission^.XPick) THEN	// Direzione NEGATIVA 
				FOR wa := WAPARTENZA TO NPOSTAZIONE_DOPORIBALTINO BY -1 DO
					AltezzaDiIngombroArea := 0;
					IF WorkAreaState^[wa].H > WorkAreaState^[wa].HPL THEN
						AltezzaDiIngombroArea := WorkAreaState^[wa].H;
					ELSE
						AltezzaDiIngombroArea := WorkAreaState^[wa].HPL;
					END_IF
					IF QuotaAnticipoDinamicaZ_VersoPrelPacco <= AltezzaDiIngombroArea + TCPParameter.Z + OffsetSicurezzaAnticipoMovimenti.OffsetSicurezzaAnticipo_Z THEN
						QuotaAnticipoDinamicaZ_VersoPrelPacco := AltezzaDiIngombroArea + TCPParameter.Z + OffsetSicurezzaAnticipoMovimenti.OffsetSicurezzaAnticipo_Z;
					END_IF
				END_FOR		
				(* Valuto I Pick-Point *)
				(*FOR P:=1 TO MAXPICKPOINT DO
					AltezzaDiIngombroPuntiPrelievo := 0;
					IF  WorkPickPoint^[P].Zh + WorkPickPointState^[P].ZDim >= WorkPickPointDimension[P].Zdim THEN // Se Altezza orrizzontale Ribaltino + Zpacco >= Ingombro Verticale Ribaltino
						AltezzaDiIngombroPuntiPrelievo := WorkPickPoint^[P].Zh + WorkPickPointState^[P].ZDim;
					END_IF
					IF WorkPickPoint^[P].Zv + WorkPickPointState^[P].ZTilter + WorkPickPointState^[P].YDim >= WorkPickPointDimension[P].Zdim THEN // Se Altezza Vertivale Ribaltino + Quota Fermo + Ypacco >= Ingombro Verticale Ribaltino
						AltezzaDiIngombroPuntiPrelievo := WorkPickPoint^[P].Zv + WorkPickPointState^[P].ZTilter + WorkPickPointState^[P].YDim;
					END_IF
					IF WorkPickPointDimension[P].Zdim >= AltezzaDiIngombroPuntiPrelievo THEN //Se Ingombro Verticale Ribaltino >= Dell'ingombro valutato sopra
						AltezzaDiIngombroPuntiPrelievo := WorkPickPointDimension[P].Zdim;
					END_IF
					IF WAPARTENZA = NPOSTAZIONE_DOPORIBALTINO THEN //Se sono nella posizione 7 valuto l'altezza del ribaltino "REALE", con o senza pacco
						IF QuotaAnticipoDinamicaZ_VersoPrelPacco <= AltezzaDiIngombroPuntiPrelievo + TCPParameter.Z + OffsetSicurezza.Avuoto THEN //Se Quota fuori ingombro <= dell' ingombro del punto di prelievo
							QuotaAnticipoDinamicaZ_VersoPrelPacco := AltezzaDiIngombroPuntiPrelievo + TCPParameter.Z + OffsetSicurezza.Avuoto;
						END_IF	
					ELSE
						IF QuotaAnticipoDinamicaZ_VersoPrelPacco <= AltezzaDiIngombroPuntiPrelievo + TCPParameter.Z + OffsetSicurezzaAnticipoMovimenti.OffsetSicurezzaAnticipo_Z - 300 THEN
							QuotaAnticipoDinamicaZ_VersoPrelPacco := AltezzaDiIngombroPuntiPrelievo + WorkPickPointState^[P].YDim + TCPParameter.Z + OffsetSicurezzaAnticipoMovimenti.OffsetSicurezzaAnticipo_Z - 300;
						END_IF
					END_IF
				END_FOR*)
			ELSE		// Direzione POSITIVA
				FOR wa := WAPARTENZA TO NPOSTAZIONE_PRIMADELPUNTODIPREL DO
					AltezzaDiIngombroArea := 0;
					IF WorkAreaState^[wa].H > WorkAreaState^[wa].HPL THEN
						AltezzaDiIngombroArea := WorkAreaState^[wa].H;
					ELSE
						AltezzaDiIngombroArea := WorkAreaState^[wa].HPL;
					END_IF
					IF QuotaAnticipoDinamicaZ_VersoPrelPacco <= AltezzaDiIngombroArea + TCPParameter.Z + OffsetSicurezzaAnticipoMovimenti.OffsetSicurezzaAnticipo_Z THEN
						QuotaAnticipoDinamicaZ_VersoPrelPacco := AltezzaDiIngombroArea + TCPParameter.Z + OffsetSicurezzaAnticipoMovimenti.OffsetSicurezzaAnticipo_Z;
					END_IF
				END_FOR			
								
				(* Valuto I Pick-Point *)
				(*FOR P:=1 TO MAXPICKPOINT DO
					AltezzaDiIngombroPuntiPrelievo := 0;
					IF  WorkPickPoint^[P].Zh + WorkPickPointState^[P].ZDim >= WorkPickPointDimension[P].Zdim THEN // Se Altezza orrizzontale Ribaltino + Zpacco >= Ingombro Verticale Ribaltino
						AltezzaDiIngombroPuntiPrelievo := WorkPickPoint^[P].Zh + WorkPickPointState^[P].ZDim;
					END_IF
					IF WorkPickPoint^[P].Zv + WorkPickPointState^[P].ZTilter + WorkPickPointState^[P].YDim >= WorkPickPointDimension[P].Zdim THEN // Se Altezza Vertivale Ribaltino + Quota Fermo + Ypacco >= Ingombro Verticale Ribaltino
						AltezzaDiIngombroPuntiPrelievo := WorkPickPoint^[P].Zv + WorkPickPointState^[P].ZTilter + WorkPickPointState^[P].YDim;
					END_IF
					IF WorkPickPointDimension[P].Zdim >= AltezzaDiIngombroPuntiPrelievo THEN //Se Ingombro Verticale Ribaltino >= Dell'ingombro valutato sopra
						AltezzaDiIngombroPuntiPrelievo := WorkPickPointDimension[P].Zdim;
					END_IF
					IF WAPARTENZA = NPOSTAZIONE_PRIMADELPUNTODIPREL THEN //Se sono nella posizione 7 valuto l'altezza del ribaltino "REALE", con o senza pacco
						IF QuotaAnticipoDinamicaZ_VersoPrelPacco <= AltezzaDiIngombroPuntiPrelievo + TCPParameter.Z + OffsetSicurezza.Avuoto THEN //Se Quota fuori ingombro <= dell' ingombro del punto di prelievo
							QuotaAnticipoDinamicaZ_VersoPrelPacco := AltezzaDiIngombroPuntiPrelievo + TCPParameter.Z + OffsetSicurezza.Avuoto;
						END_IF
					ELSE		//Se non sono nella WA 7, do una quota fittizzia, inferiore all'altezza del ribaltino "reale"
						IF QuotaAnticipoDinamicaZ_VersoPrelPacco <= AltezzaDiIngombroPuntiPrelievo + TCPParameter.Z + OffsetSicurezzaAnticipoMovimenti.OffsetSicurezzaAnticipo_Z - 300 THEN
							QuotaAnticipoDinamicaZ_VersoPrelPacco := AltezzaDiIngombroPuntiPrelievo + WorkPickPointState^[P].YDim + TCPParameter.Z + OffsetSicurezzaAnticipoMovimenti.OffsetSicurezzaAnticipo_Z - 300;
						END_IF
					END_IF
				END_FOR	*)
			END_IF
				IF ModuleAX_Z^.Ax^.Status.ActPosition >= QuotaAnticipoDinamicaZ_VersoPrelPacco THEN
					QuotaAnticipoDinamicaZ_Raggiunta := TRUE;
				ELSE
					QuotaAnticipoDinamicaZ_Raggiunta := FALSE;
				END_IF
		END_IF
	
				
	WAMANAGER_CICLO_PRELIEVO_PACCO_END,
		
	WAMANAGER_CICLO_DEPOSITO_PACCO_RUN:
		(*IF AbilitaAnticipoDinamico AND Forming^[WorkAreaState^[Mission^.PPlace].F].PackXN[WorkAreaState^[Mission^.PPlace].P].Trajectory <> 2 AND
	    	Forming^[WorkAreaState^[Mission^.PPlace].F].PackXN[WorkAreaState^[Mission^.PPlace].P].Trajectory <> 101 AND
			Forming^[WorkAreaState^[Mission^.PPlace].F].PackXN[WorkAreaState^[Mission^.PPlace].P].Trajectory <> 201 AND
			Forming^[WorkAreaState^[Mission^.PPlace].F].PackXP[WorkAreaState^[Mission^.PPlace].P].Trajectory <> 101 AND
			Forming^[WorkAreaState^[Mission^.PPlace].F].PackXP[WorkAreaState^[Mission^.PPlace].P].Trajectory <> 201 THEN
			QuotaAnticipoDinamicaX_DepositoPacco := 0;
			
			
			//IF DirezioneXPositiva_Dep THEN
			IF NOT TFDirezioneAssePositiva(Posizione_Attuale:=ModuleAX_X^.Ax^.Status.ActPosition,Posizione_Finale:=Mission^.XPlace) THEN
				IF Mission^.PPlace < NPOSTAZIONE_PRIMADELPUNTODIPREL THEN
					IF WorkAreaState^[Mission^.PPlace + 1].P <= 1 THEN
						QuotaAnticipoDinamicaX_DepositoPacco := (Workarea^[Mission^.PPlace + 1].X - Pallet^[Workarea^[Mission^.PPlace + 1].Pallet].X/2 + OffsetSicurezzaAnticipoMovimenti.OffsetSicurezzaAnticipo_X + (IngombroX/2));
					ELSE
						QuotaAnticipoDinamicaX_DepositoPacco := (Workarea^[Mission^.PPlace + 1].X + Pallet^[Workarea^[Mission^.PPlace + 1].Pallet].X/2 + OffsetSicurezzaAnticipoMovimenti.OffsetSicurezzaAnticipo_X + (IngombroX/2));
					END_IF	
				ELSIF Mission^.PPlace > NPOSTAZIONE_DOPORIBALTINO THEN
					IF WorkAreaState^[Mission^.PPlace + 1].P <= 1 THEN
						QuotaAnticipoDinamicaX_DepositoPacco := (Workarea^[Mission^.PPlace + 1].X - Pallet^[Workarea^[Mission^.PPlace + 1].Pallet].X/2 + OffsetSicurezzaAnticipoMovimenti.OffsetSicurezzaAnticipo_X + (IngombroX/2));
					ELSE
						QuotaAnticipoDinamicaX_DepositoPacco := (Workarea^[Mission^.PPlace + 1].X + Pallet^[Workarea^[Mission^.PPlace + 1].Pallet].X/2 + OffsetSicurezzaAnticipoMovimenti.OffsetSicurezzaAnticipo_X + (IngombroX/2));
					END_IF
					//IF QuotaAnticipoDinamicaX_DepositoPacco <= Workarea^[NPOSTAZIONE_DOPORIBALTINO].X + 800 + (IngombroX/2) + OffsetSicurezzaAnticipoMovimenti.OffsetSicurezzaAnticipo_X THEN
					//	QuotaAnticipoDinamicaX_DepositoPacco := Workarea^[NPOSTAZIONE_DOPORIBALTINO].X + 800 + (IngombroX/2) + OffsetSicurezzaAnticipoMovimenti.OffsetSicurezzaAnticipo_X;
					//END_IF
				ELSIF Mission^.PPlace = NPOSTAZIONE_DOPORIBALTINO OR Mission^.PPlace = NPOSTAZIONE_PRIMADELPUNTODIPREL THEN //postazione 5,6
					QuotaAnticipoDinamicaX_DepositoPacco := (WorkPickPoint^[Mission^.PPick].Xv + LarghezzaPickPoint/2 + OffsetSicurezzaAnticipoMovimenti.OffsetSicurezzaAnticipo_X + (IngombroX/2));
				END_IF
				IF ModuleAX_X^.Ax^.Status.ActPosition <= QuotaAnticipoDinamicaX_DepositoPacco THEN
					QuotaAnticipoDinamicaX_Raggiunta := TRUE;
				ELSE
					QuotaAnticipoDinamicaX_Raggiunta := FALSE;
				END_IF
				TFCalcolaNumeroPostazioneDXSX(PosizioneAttuale	:= ModuleAX_X^.Ax^.Status.ActPosition,
												WorkArea		:= WorkArea,
												DirezioneAsseX_Positiva := FALSE,
												NPostazioneDX	=> WADX,
												NPostazioneSX	=> WASX,
												PostazionePartenza=>WAPARTENZA);
			ELSE	//Direzione POSITIVA
				IF Mission^.PPlace < NPOSTAZIONE_PRIMADELPUNTODIPREL OR Mission^.PPlace > NPOSTAZIONE_DOPORIBALTINO THEN
					IF WorkAreaState^[Mission^.PPlace - 1].P <= 1 OR WorkArea^[Mission^.PPlace - 1].H + 100 < WorkArea^[Mission^.PPlace].H  THEN
						QuotaAnticipoDinamicaX_DepositoPacco := (Workarea^[Mission^.PPlace - 1].X + Pallet^[Workarea^[Mission^.PPlace - 1].Pallet].X/2 - OffsetSicurezzaAnticipoMovimenti.OffsetSicurezzaAnticipo_X - (IngombroX/2));
					ELSE
						QuotaAnticipoDinamicaX_DepositoPacco := (Workarea^[Mission^.PPlace - 1].X - Pallet^[Workarea^[Mission^.PPlace - 1].Pallet].X/2 - OffsetSicurezzaAnticipoMovimenti.OffsetSicurezzaAnticipo_X - (IngombroX/2));
					END_IF
				ELSIF Mission^.PPlace = NPOSTAZIONE_PRIMADELPUNTODIPREL OR  Mission^.PPlace = NPOSTAZIONE_DOPORIBALTINO THEN
					QuotaAnticipoDinamicaX_DepositoPacco := (WorkPickPoint^[Mission^.PPick].Xv - LarghezzaPickPoint/2 - OffsetSicurezzaAnticipoMovimenti.OffsetSicurezzaAnticipo_X - (IngombroX/2));
				END_IF
				IF ModuleAX_X^.Ax^.Status.ActPosition >= QuotaAnticipoDinamicaX_DepositoPacco THEN
					QuotaAnticipoDinamicaX_Raggiunta := TRUE;
				ELSE
					QuotaAnticipoDinamicaX_Raggiunta := FALSE;
				END_IF
				TFCalcolaNumeroPostazioneDXSX(PosizioneAttuale	:= ModuleAX_X^.Ax^.Status.ActPosition,
												WorkArea		:= WorkArea,
												DirezioneAsseX_Positiva := TRUE,
												NPostazioneDX	=> WADX,
												NPostazioneSX	=> WASX,
												PostazionePartenza=>WAPARTENZA);
			END_IF
		END_IF*)
		
		WAPARTENZA := Mission^.PPlace;
				
	//WAMANAGER_CICLO_DEPOSITO_PACCO_END;
	*)
END_CASE

END_FUNCTION_BLOCK

// ---- POUs/TFPalletizerDataTF/TFValutaAssiInFinestraDiPassMode.TcPOU
FUNCTION_BLOCK TFValutaAssiInFinestraDiPassMode
VAR_INPUT
	ModuleAX_X : POINTER TO TFModulePalletizer_Ax;
	ModuleAX_Y : POINTER TO TFModulePalletizer_Ax;
	ModuleAX_Z : POINTER TO TFModulePalletizer_Ax;
	ModuleAX_J : POINTER TO TFModulePalletizer_AxJ_Lastre;
	Traiettoria : POINTER TO TFTraiettoria;
	WorkAreaManager : POINTER TO TFWorkAreaManager;
END_VAR
VAR
	Direzione_X_Positiva : BOOL;
	Direzione_Y_Positiva : BOOL;
	Direzione_Z_Positiva : BOOL;
	Direzione_J_Positiva : BOOL;
	Direzione_K_Positiva : bool;
	AsseXInMoto: BOOL;
	AsseYInMoto: BOOL;
	AsseZInMoto: BOOL;
	AsseJInMoto: BOOL;
	//AsseKInMoto: BOOL;
	OffsetPassModeY_Appoggio: REAL;
END_VAR

(* Azzero le variabili *)
Asse_X_InFinestraDiPassMode := FALSE;
Asse_Y_InFinestraDiPassMode := FALSE;
Asse_Z_InFinestraDiPassMode := FALSE;
Asse_J_InFinestraDiPassMode := FALSE;

(* Valuto la direzione degli assi *)
Direzione_X_Positiva := TFDirezioneAssePositiva(Posizione_Attuale:=ModuleAX_X^.Ax^.Status.ActPosition,Posizione_Finale:=ProgrammaToModule_X.Quota_Destinazione);
Direzione_Y_Positiva := TFDirezioneAssePositiva(Posizione_Attuale:=ModuleAX_Y^.Ax^.Status.ActPosition,Posizione_Finale:=ProgrammaToModule_Y.Quota_Destinazione);
Direzione_Z_Positiva := TFDirezioneAssePositiva(Posizione_Attuale:=ModuleAX_Z^.Ax^.Status.ActPosition,Posizione_Finale:=ProgrammaToModule_Z.Quota_Destinazione);
Direzione_J_Positiva := TFDirezioneAssePositiva(Posizione_Attuale:=ModuleAX_J^.Ax^.Status.ActPosition,Posizione_Finale:=ProgrammaToModule_J.Quota_Destinazione);
(* Valuto se gli assi si stanno muovendo *)
AsseXInMoto:=ModuleAX_X^.Ax^.AxRef^.Status.Moving;
AsseYInMoto:=ModuleAX_Y^.Ax^.AxRef^.Status.Moving;
AsseZInMoto:=ModuleAX_Z^.Ax^.AxRef^.Status.Moving;
AsseJInMoto:=ModuleAX_J^.Ax^.AxRef^.Status.Moving;

IF Traiettoria^.PassModeGlobalEnable AND AbilitazionePassModeGlobale THEN (* Abilitazione Globale del PassMode*)
	
//	CASE WorkAreaManager^.State OF
		
//		WAMANAGER_CICLO_RIPOSO_RUN: 
			(* Abilito tutti i pasmode*)
			Traiettoria^.PassModePoint_X_Enable[1] := TRUE; 
			Traiettoria^.PassModePoint_Y_Enable[1] := TRUE; 
			Traiettoria^.PassModePoint_Z_Enable[1] := TRUE;
			Traiettoria^.PassModePoint_J_Enable[1] := TRUE;
			Traiettoria^.PassModePoint_K_Enable[1] := TRUE;
			(* Valuta il Pass Mode Per L'asse X *)
			IF Traiettoria^.PassModePoint_X_Enable[1] THEN
				IF AsseXInMoto THEN
					IF Direzione_X_Positiva THEN	//Se l'asse si sta muovendo in direzione POSITIVA
						IF ModuleAX_X^.Ax^.Status.ActPosition >= (ProgrammaToModule_X.Quota_Destinazione - OffsetPassMode.X) THEN
							Asse_X_InFinestraDiPassMode := TRUE;	
						END_IF
					ELSE							//Se l'asse si sta muovendo in direzione NEGATIVA
						IF ModuleAX_X^.Ax^.Status.ActPosition <= (ProgrammaToModule_X.Quota_Destinazione + OffsetPassMode.X) THEN
							Asse_X_InFinestraDiPassMode := TRUE;	
						END_IF
					END_IF
				END_IF
			END_IF
				
			(* Valuta il Pass Mode Per L'asse Y *)
			IF Traiettoria^.PassModePoint_Y_Enable[1] THEN
				IF Pinza_InIngombroColonne_Attuale THEN
					OffsetPassModeY_Appoggio := 80;
				ELSE
					OffsetPassModeY_Appoggio := OffsetPassMode.Y;
				END_IF
				IF AsseYInMoto THEN
					IF Direzione_Y_Positiva THEN	//Se l'asse si sta muovendo in direzione POSITIVA
						IF ModuleAX_Y^.Ax^.Status.ActPosition >= (ProgrammaToModule_Y.Quota_Destinazione - OffsetPassModeY_Appoggio) THEN
							Asse_Y_InFinestraDiPassMode := TRUE;	
						END_IF
					ELSE							//Se l'asse si sta muovendo in direzione NEGATIVA
						IF ModuleAX_Y^.Ax^.Status.ActPosition <= (ProgrammaToModule_Y.Quota_Destinazione + OffsetPassModeY_Appoggio) THEN
							Asse_Y_InFinestraDiPassMode := TRUE;	
						END_IF
					END_IF
				END_IF
			END_IF
			
			(* Valuta il Pass Mode Per L'asse Z *)
			IF Traiettoria^.PassModePoint_Z_Enable[1] THEN
				IF AsseZInMoto THEN
					IF Direzione_Z_Positiva THEN	//Se l'asse si sta muovendo in direzione POSITIVA
						IF ModuleAX_Z^.Ax^.Status.ActPosition >= (ProgrammaToModule_Z.Quota_Destinazione - OffsetPassMode.Z) THEN
							Asse_Z_InFinestraDiPassMode := TRUE;	
						END_IF
					ELSE							//Se l'asse si sta muovendo in direzione NEGATIVA
						IF ModuleAX_Z^.Ax^.Status.ActPosition <= (ProgrammaToModule_Z.Quota_Destinazione + OffsetPassMode.Z) THEN
							Asse_Z_InFinestraDiPassMode := TRUE;	
						END_IF
					END_IF
				END_IF
			END_IF
			
			(* Valuta il Pass Mode Per L'asse J *)
			IF Traiettoria^.PassModePoint_J_Enable[1] THEN
				IF AsseJInMoto THEN
					IF Direzione_J_Positiva THEN	//Se l'asse si sta muovendo in direzione POSITIVA
						IF ModuleAX_J^.Ax^.Status.ActPosition >= (ProgrammaToModule_J.Quota_Destinazione - OffsetPassMode.J) THEN
							Asse_J_InFinestraDiPassMode := TRUE;	
						END_IF
					ELSE							//Se l'asse si sta muovendo in direzione NEGATIVA
						IF ModuleAX_J^.Ax^.Status.ActPosition <= (ProgrammaToModule_J.Quota_Destinazione + OffsetPassMode.J) THEN
							Asse_J_InFinestraDiPassMode := TRUE;	
						END_IF
					END_IF
				END_IF
			END_IF
		(*
		WAMANAGER_CICLO_PRELIEVO_PALL_RUN: 
			(* Abilito tutti i pasmode*)
			Traiettoria^.PassModePoint_X_Enable[1] := TRUE; 
			Traiettoria^.PassModePoint_Y_Enable[1] := TRUE; 
			Traiettoria^.PassModePoint_Z_Enable[1] := TRUE;
			Traiettoria^.PassModePoint_J_Enable[1] := TRUE;
			Traiettoria^.PassModePoint_K_Enable[1] := TRUE;
			(* Valuta il Pass Mode Per L'asse X *)
			IF Traiettoria^.PassModePoint_X_Enable[1] THEN
				IF AsseXInMoto THEN
					IF Direzione_X_Positiva THEN	//Se l'asse si sta muovendo in direzione POSITIVA
						IF ModuleAX_X^.Ax^.Status.ActPosition >= (ProgrammaToModule_X.Quota_Destinazione - OffsetPassMode.X) THEN
							Asse_X_InFinestraDiPassMode := TRUE;	
						END_IF
					ELSE							//Se l'asse si sta muovendo in direzione NEGATIVA
						IF ModuleAX_X^.Ax^.Status.ActPosition <= (ProgrammaToModule_X.Quota_Destinazione + OffsetPassMode.X) THEN
							Asse_X_InFinestraDiPassMode := TRUE;	
						END_IF
					END_IF
				END_IF
			END_IF
				
			(* Valuta il Pass Mode Per L'asse Y *)
			IF Traiettoria^.PassModePoint_Y_Enable[1] THEN
				IF AsseYInMoto THEN
					IF Pinza_InIngombroColonne_Attuale THEN
						OffsetPassModeY_Appoggio := 80;
					ELSE
						OffsetPassModeY_Appoggio := OffsetPassMode.Y;
					END_IF
					IF Direzione_Y_Positiva THEN	//Se l'asse si sta muovendo in direzione POSITIVA
						IF ModuleAX_Y^.Ax^.Status.ActPosition >= (ProgrammaToModule_Y.Quota_Destinazione - OffsetPassModeY_Appoggio) THEN
							Asse_Y_InFinestraDiPassMode := TRUE;	
						END_IF
					ELSE							//Se l'asse si sta muovendo in direzione NEGATIVA
						IF ModuleAX_Y^.Ax^.Status.ActPosition <= (ProgrammaToModule_Y.Quota_Destinazione + OffsetPassModeY_Appoggio) THEN
							Asse_Y_InFinestraDiPassMode := TRUE;	
						END_IF
					END_IF	
				END_IF
			END_IF
			
			(* Valuta il Pass Mode Per L'asse Z *)
			IF Traiettoria^.PassModePoint_Z_Enable[1] THEN
				IF AsseZInMoto THEN
					IF Direzione_Z_Positiva THEN	//Se l'asse si sta muovendo in direzione POSITIVA
						IF ModuleAX_Z^.Ax^.Status.ActPosition >= (ProgrammaToModule_Z.Quota_Destinazione - OffsetPassMode.Z) THEN
							Asse_Z_InFinestraDiPassMode := TRUE;	
						END_IF
					ELSE							//Se l'asse si sta muovendo in direzione NEGATIVA
						IF ModuleAX_Z^.Ax^.Status.ActPosition <= (ProgrammaToModule_Z.Quota_Destinazione + OffsetPassMode.Z) THEN
							Asse_Z_InFinestraDiPassMode := TRUE;	
						END_IF
					END_IF
				END_IF
			END_IF
			
			(* Valuta il Pass Mode Per L'asse J *)
			IF Traiettoria^.PassModePoint_J_Enable[1] THEN
				IF AsseJInMoto THEN
					IF Direzione_J_Positiva THEN	//Se l'asse si sta muovendo in direzione POSITIVA
						IF ModuleAX_J^.Ax^.Status.ActPosition >= (ProgrammaToModule_J.Quota_Destinazione - OffsetPassMode.J) THEN
							Asse_J_InFinestraDiPassMode := TRUE;	
						END_IF
					ELSE							//Se l'asse si sta muovendo in direzione NEGATIVA
						IF ModuleAX_J^.Ax^.Status.ActPosition <= (ProgrammaToModule_J.Quota_Destinazione + OffsetPassMode.J) THEN
							Asse_J_InFinestraDiPassMode := TRUE;	
						END_IF
					END_IF
				END_IF
			END_IF
									
		WAMANAGER_CICLO_DEPOSITO_PALL_RUN: 
			(* Abilito tutti i pasmode*)
			Traiettoria^.PassModePoint_X_Enable[1] := TRUE; 
			Traiettoria^.PassModePoint_Y_Enable[1] := TRUE; 
			Traiettoria^.PassModePoint_Z_Enable[1] := TRUE;
			Traiettoria^.PassModePoint_J_Enable[1] := TRUE;
			Traiettoria^.PassModePoint_K_Enable[1] := TRUE;
			(* Valuta il Pass Mode Per L'asse X *)
			IF Traiettoria^.PassModePoint_X_Enable[1] THEN
				IF AsseXInMoto THEN
					IF Direzione_X_Positiva THEN	//Se l'asse si sta muovendo in direzione POSITIVA
						IF ModuleAX_X^.Ax^.Status.ActPosition >= (ProgrammaToModule_X.Quota_Destinazione - OffsetPassMode.X) THEN
							Asse_X_InFinestraDiPassMode := TRUE;	
						END_IF
					ELSE							//Se l'asse si sta muovendo in direzione NEGATIVA
						IF ModuleAX_X^.Ax^.Status.ActPosition <= (ProgrammaToModule_X.Quota_Destinazione + OffsetPassMode.X) THEN
							Asse_X_InFinestraDiPassMode := TRUE;	
						END_IF
					END_IF
				END_IF
			END_IF
				
			(* Valuta il Pass Mode Per L'asse Y *)
			IF Traiettoria^.PassModePoint_Y_Enable[1] THEN
				IF AsseYInMoto THEN
					IF Direzione_Y_Positiva THEN	//Se l'asse si sta muovendo in direzione POSITIVA
						IF ModuleAX_Y^.Ax^.Status.ActPosition >= (ProgrammaToModule_Y.Quota_Destinazione - OffsetPassMode.Y) THEN
							Asse_Y_InFinestraDiPassMode := TRUE;	
						END_IF
					ELSE							//Se l'asse si sta muovendo in direzione NEGATIVA
						IF ModuleAX_Y^.Ax^.Status.ActPosition <= (ProgrammaToModule_Y.Quota_Destinazione + OffsetPassMode.Y) THEN
							Asse_Y_InFinestraDiPassMode := TRUE;	
						END_IF
					END_IF
				END_IF
			END_IF
			
			(* Valuta il Pass Mode Per L'asse Z *)
			IF Traiettoria^.PassModePoint_Z_Enable[1] THEN
				IF AsseZInMoto THEN
					IF Direzione_Z_Positiva THEN	//Se l'asse si sta muovendo in direzione POSITIVA
						IF ModuleAX_Z^.Ax^.Status.ActPosition >= (ProgrammaToModule_Z.Quota_Destinazione - OffsetPassMode.Z) THEN
							Asse_Z_InFinestraDiPassMode := TRUE;	
						END_IF
					ELSE							//Se l'asse si sta muovendo in direzione NEGATIVA
						IF ModuleAX_Z^.Ax^.Status.ActPosition <= (ProgrammaToModule_Z.Quota_Destinazione + OffsetPassMode.Z) THEN
							Asse_Z_InFinestraDiPassMode := TRUE;	
						END_IF
					END_IF
				END_IF
			END_IF
			
			(* Valuta il Pass Mode Per L'asse J *)
			IF Traiettoria^.PassModePoint_J_Enable[1] THEN
				IF AsseJInMoto THEN
					IF Direzione_J_Positiva THEN	//Se l'asse si sta muovendo in direzione POSITIVA
						IF ModuleAX_J^.Ax^.Status.ActPosition >= (ProgrammaToModule_J.Quota_Destinazione - OffsetPassMode.J) THEN
							Asse_J_InFinestraDiPassMode := TRUE;	
						END_IF
					ELSE							//Se l'asse si sta muovendo in direzione NEGATIVA
						IF ModuleAX_J^.Ax^.Status.ActPosition <= (ProgrammaToModule_J.Quota_Destinazione + OffsetPassMode.J) THEN
							Asse_J_InFinestraDiPassMode := TRUE;	
						END_IF
					END_IF
				END_IF
			END_IF
									
		WAMANAGER_CICLO_PRELIEVO_FALDA_VUOTI_RUN:
			(* Abilito tutti i pasmode*)
			Traiettoria^.PassModePoint_X_Enable[1] := TRUE; 
			Traiettoria^.PassModePoint_Y_Enable[1] := TRUE; 
			Traiettoria^.PassModePoint_Z_Enable[1] := TRUE;
			Traiettoria^.PassModePoint_J_Enable[1] := TRUE;
			Traiettoria^.PassModePoint_K_Enable[1] := TRUE;
			(* Valuta il Pass Mode Per L'asse X *)
			IF Traiettoria^.PassModePoint_X_Enable[1] THEN
				IF AsseXInMoto THEN
					IF Direzione_X_Positiva THEN	//Se l'asse si sta muovendo in direzione POSITIVA
						IF ModuleAX_X^.Ax^.Status.ActPosition >= (ProgrammaToModule_X.Quota_Destinazione - OffsetPassMode.X) THEN
							Asse_X_InFinestraDiPassMode := TRUE;	
						END_IF
					ELSE							//Se l'asse si sta muovendo in direzione NEGATIVA
						IF ModuleAX_X^.Ax^.Status.ActPosition <= (ProgrammaToModule_X.Quota_Destinazione + OffsetPassMode.X) THEN
							Asse_X_InFinestraDiPassMode := TRUE;	
						END_IF
					END_IF
				END_IF
			END_IF
				
			(* Valuta il Pass Mode Per L'asse Y *)
			IF Traiettoria^.PassModePoint_Y_Enable[1] THEN
				IF Pinza_InIngombroColonne_Attuale THEN
					OffsetPassModeY_Appoggio := 80;
				ELSE
					OffsetPassModeY_Appoggio := OffsetPassMode.Y;
				END_IF
				IF AsseYInMoto THEN
					IF Direzione_Y_Positiva THEN	//Se l'asse si sta muovendo in direzione POSITIVA
						IF ModuleAX_Y^.Ax^.Status.ActPosition >= (ProgrammaToModule_Y.Quota_Destinazione - OffsetPassModeY_Appoggio) THEN
							Asse_Y_InFinestraDiPassMode := TRUE;	
						END_IF
					ELSE							//Se l'asse si sta muovendo in direzione NEGATIVA
						IF ModuleAX_Y^.Ax^.Status.ActPosition <= (ProgrammaToModule_Y.Quota_Destinazione + OffsetPassModeY_Appoggio) THEN
							Asse_Y_InFinestraDiPassMode := TRUE;	
						END_IF
					END_IF
				END_IF
			END_IF
			
			(* Valuta il Pass Mode Per L'asse Z *)
			IF Traiettoria^.PassModePoint_Z_Enable[1] THEN
				IF AsseZInMoto THEN
					IF Direzione_Z_Positiva THEN	//Se l'asse si sta muovendo in direzione POSITIVA
						IF ModuleAX_Z^.Ax^.Status.ActPosition >= (ProgrammaToModule_Z.Quota_Destinazione - OffsetPassMode.Z) THEN
							Asse_Z_InFinestraDiPassMode := TRUE;	
						END_IF
					ELSE							//Se l'asse si sta muovendo in direzione NEGATIVA
						IF ModuleAX_Z^.Ax^.Status.ActPosition <= (ProgrammaToModule_Z.Quota_Destinazione + OffsetPassMode.Z) THEN
							Asse_Z_InFinestraDiPassMode := TRUE;	
						END_IF
					END_IF
				END_IF
			END_IF
			
			(* Valuta il Pass Mode Per L'asse J *)
			IF Traiettoria^.PassModePoint_J_Enable[1] THEN
				IF AsseJInMoto THEN
					IF Direzione_J_Positiva THEN	//Se l'asse si sta muovendo in direzione POSITIVA
						IF ModuleAX_J^.Ax^.Status.ActPosition >= (ProgrammaToModule_J.Quota_Destinazione - OffsetPassMode.J) THEN
							Asse_J_InFinestraDiPassMode := TRUE;	
						END_IF
					ELSE							//Se l'asse si sta muovendo in direzione NEGATIVA
						IF ModuleAX_J^.Ax^.Status.ActPosition <= (ProgrammaToModule_J.Quota_Destinazione + OffsetPassMode.J) THEN
							Asse_J_InFinestraDiPassMode := TRUE;	
						END_IF
					END_IF
				END_IF
			END_IF
									
		WAMANAGER_CICLO_DEPOSITO_FALDA_VUOTI_RUN:
			(* Abilito tutti i pasmode*)
			Traiettoria^.PassModePoint_X_Enable[1] := TRUE; 
			Traiettoria^.PassModePoint_Y_Enable[1] := TRUE; 
			Traiettoria^.PassModePoint_Z_Enable[1] := TRUE;
			Traiettoria^.PassModePoint_J_Enable[1] := TRUE;
			Traiettoria^.PassModePoint_K_Enable[1] := TRUE;
			(* Valuta il Pass Mode Per L'asse X *)
			IF Traiettoria^.PassModePoint_X_Enable[1] THEN
				IF AsseXInMoto THEN
					IF Direzione_X_Positiva THEN	//Se l'asse si sta muovendo in direzione POSITIVA
						IF ModuleAX_X^.Ax^.Status.ActPosition >= (ProgrammaToModule_X.Quota_Destinazione - OffsetPassMode.X) THEN
							Asse_X_InFinestraDiPassMode := TRUE;	
						END_IF
					ELSE							//Se l'asse si sta muovendo in direzione NEGATIVA
						IF ModuleAX_X^.Ax^.Status.ActPosition <= (ProgrammaToModule_X.Quota_Destinazione + OffsetPassMode.X) THEN
							Asse_X_InFinestraDiPassMode := TRUE;	
						END_IF
					END_IF
				END_IF
			END_IF
				
			(* Valuta il Pass Mode Per L'asse Y *)
			IF Traiettoria^.PassModePoint_Y_Enable[1] THEN
				IF AsseYInMoto THEN
					IF Direzione_Y_Positiva THEN	//Se l'asse si sta muovendo in direzione POSITIVA
						IF ModuleAX_Y^.Ax^.Status.ActPosition >= (ProgrammaToModule_Y.Quota_Destinazione - OffsetPassMode.Y) THEN
							Asse_Y_InFinestraDiPassMode := TRUE;	
						END_IF
					ELSE							//Se l'asse si sta muovendo in direzione NEGATIVA
						IF ModuleAX_Y^.Ax^.Status.ActPosition <= (ProgrammaToModule_Y.Quota_Destinazione + OffsetPassMode.Y) THEN
							Asse_Y_InFinestraDiPassMode := TRUE;	
						END_IF
					END_IF
				END_IF
			END_IF
			
			(* Valuta il Pass Mode Per L'asse Z *)
			IF Traiettoria^.PassModePoint_Z_Enable[1] THEN
				IF AsseZInMoto THEN
					IF Direzione_Z_Positiva THEN	//Se l'asse si sta muovendo in direzione POSITIVA
						IF ModuleAX_Z^.Ax^.Status.ActPosition >= (ProgrammaToModule_Z.Quota_Destinazione - OffsetPassMode.Z) THEN
							Asse_Z_InFinestraDiPassMode := TRUE;	
						END_IF
					ELSE							//Se l'asse si sta muovendo in direzione NEGATIVA
						IF ModuleAX_Z^.Ax^.Status.ActPosition <= (ProgrammaToModule_Z.Quota_Destinazione + OffsetPassMode.Z) THEN
							Asse_Z_InFinestraDiPassMode := TRUE;	
						END_IF
					END_IF
				END_IF
			END_IF
			
			(* Valuta il Pass Mode Per L'asse J *)
			IF Traiettoria^.PassModePoint_J_Enable[1] THEN
				IF AsseJInMoto THEN
					IF Direzione_J_Positiva THEN	//Se l'asse si sta muovendo in direzione POSITIVA
						IF ModuleAX_J^.Ax^.Status.ActPosition >= (ProgrammaToModule_J.Quota_Destinazione - OffsetPassMode.J) THEN
							Asse_J_InFinestraDiPassMode := TRUE;	
						END_IF
					ELSE							//Se l'asse si sta muovendo in direzione NEGATIVA
						IF ModuleAX_J^.Ax^.Status.ActPosition <= (ProgrammaToModule_J.Quota_Destinazione + OffsetPassMode.J) THEN
							Asse_J_InFinestraDiPassMode := TRUE;	
						END_IF
					END_IF
				END_IF
			END_IF
		
		WAMANAGER_CICLO_PRELIEVO_FALDA_RUN:
			(* Abilito tutti i pasmode*)
			Traiettoria^.PassModePoint_X_Enable[1] := TRUE; 
			Traiettoria^.PassModePoint_Y_Enable[1] := TRUE; 
			Traiettoria^.PassModePoint_Z_Enable[1] := TRUE;
			Traiettoria^.PassModePoint_J_Enable[1] := TRUE;
			Traiettoria^.PassModePoint_K_Enable[1] := TRUE;
			(* Valuta il Pass Mode Per L'asse X *)
			IF Traiettoria^.PassModePoint_X_Enable[1] THEN
				IF AsseXInMoto THEN
					IF Direzione_X_Positiva THEN	//Se l'asse si sta muovendo in direzione POSITIVA
						IF ModuleAX_X^.Ax^.Status.ActPosition >= (ProgrammaToModule_X.Quota_Destinazione - OffsetPassMode.X) THEN
							Asse_X_InFinestraDiPassMode := TRUE;	
						END_IF
					ELSE							//Se l'asse si sta muovendo in direzione NEGATIVA
						IF ModuleAX_X^.Ax^.Status.ActPosition <= (ProgrammaToModule_X.Quota_Destinazione + OffsetPassMode.X) THEN
							Asse_X_InFinestraDiPassMode := TRUE;	
						END_IF
					END_IF
				END_IF
			END_IF
				
			(* Valuta il Pass Mode Per L'asse Y *)
			IF Traiettoria^.PassModePoint_Y_Enable[1] THEN
				IF Pinza_InIngombroColonne_Attuale THEN
					OffsetPassModeY_Appoggio := 80;
				ELSE
					OffsetPassModeY_Appoggio := OffsetPassMode.Y;
				END_IF
				IF AsseYInMoto THEN
					IF Direzione_Y_Positiva THEN	//Se l'asse si sta muovendo in direzione POSITIVA
						IF ModuleAX_Y^.Ax^.Status.ActPosition >= (ProgrammaToModule_Y.Quota_Destinazione - OffsetPassModeY_Appoggio) THEN
							Asse_Y_InFinestraDiPassMode := TRUE;	
						END_IF
					ELSE							//Se l'asse si sta muovendo in direzione NEGATIVA
						IF ModuleAX_Y^.Ax^.Status.ActPosition <= (ProgrammaToModule_Y.Quota_Destinazione + OffsetPassModeY_Appoggio) THEN
							Asse_Y_InFinestraDiPassMode := TRUE;	
						END_IF
					END_IF
				END_IF
			END_IF
			
			(* Valuta il Pass Mode Per L'asse Z *)
			IF Traiettoria^.PassModePoint_Z_Enable[1] THEN
				IF AsseZInMoto THEN
					IF Direzione_Z_Positiva THEN	//Se l'asse si sta muovendo in direzione POSITIVA
						IF ModuleAX_Z^.Ax^.Status.ActPosition >= (ProgrammaToModule_Z.Quota_Destinazione - OffsetPassMode.Z) THEN
							Asse_Z_InFinestraDiPassMode := TRUE;	
						END_IF
					ELSE							//Se l'asse si sta muovendo in direzione NEGATIVA
						IF ModuleAX_Z^.Ax^.Status.ActPosition <= (ProgrammaToModule_Z.Quota_Destinazione + OffsetPassMode.Z) THEN
							Asse_Z_InFinestraDiPassMode := TRUE;	
						END_IF
					END_IF
				END_IF
			END_IF
			
			(* Valuta il Pass Mode Per L'asse J *)
			IF Traiettoria^.PassModePoint_J_Enable[1] THEN
				IF AsseJInMoto THEN
					IF Direzione_J_Positiva THEN	//Se l'asse si sta muovendo in direzione POSITIVA
						IF ModuleAX_J^.Ax^.Status.ActPosition >= (ProgrammaToModule_J.Quota_Destinazione - OffsetPassMode.J) THEN
							Asse_J_InFinestraDiPassMode := TRUE;	
						END_IF
					ELSE							//Se l'asse si sta muovendo in direzione NEGATIVA
						IF ModuleAX_J^.Ax^.Status.ActPosition <= (ProgrammaToModule_J.Quota_Destinazione + OffsetPassMode.J) THEN
							Asse_J_InFinestraDiPassMode := TRUE;	
						END_IF
					END_IF
				END_IF
			END_IF
			
		WAMANAGER_CICLO_DEPOSITO_FALDA_RUN:
			(* Abilito tutti i pasmode*)
			Traiettoria^.PassModePoint_X_Enable[1] := TRUE; 
			Traiettoria^.PassModePoint_Y_Enable[1] := TRUE; 
			Traiettoria^.PassModePoint_Z_Enable[1] := TRUE;
			Traiettoria^.PassModePoint_J_Enable[1] := TRUE;
			Traiettoria^.PassModePoint_K_Enable[1] := TRUE;
			(* Valuta il Pass Mode Per L'asse X *)
			IF Traiettoria^.PassModePoint_X_Enable[1] THEN
				IF AsseXInMoto THEN
					IF Direzione_X_Positiva THEN	//Se l'asse si sta muovendo in direzione POSITIVA
						IF ModuleAX_X^.Ax^.Status.ActPosition >= (ProgrammaToModule_X.Quota_Destinazione - OffsetPassMode.X) THEN
							Asse_X_InFinestraDiPassMode := TRUE;	
						END_IF
					ELSE							//Se l'asse si sta muovendo in direzione NEGATIVA
						IF ModuleAX_X^.Ax^.Status.ActPosition <= (ProgrammaToModule_X.Quota_Destinazione + OffsetPassMode.X) THEN
							Asse_X_InFinestraDiPassMode := TRUE;	
						END_IF
					END_IF
				END_IF
			END_IF
				
			(* Valuta il Pass Mode Per L'asse Y *)
			IF Traiettoria^.PassModePoint_Y_Enable[1] THEN
				IF AsseYInMoto THEN
					IF Direzione_Y_Positiva THEN	//Se l'asse si sta muovendo in direzione POSITIVA
						IF ModuleAX_Y^.Ax^.Status.ActPosition >= (ProgrammaToModule_Y.Quota_Destinazione - OffsetPassMode.Y) THEN
							Asse_Y_InFinestraDiPassMode := TRUE;	
						END_IF
					ELSE							//Se l'asse si sta muovendo in direzione NEGATIVA
						IF ModuleAX_Y^.Ax^.Status.ActPosition <= (ProgrammaToModule_Y.Quota_Destinazione + OffsetPassMode.Y) THEN
							Asse_Y_InFinestraDiPassMode := TRUE;	
						END_IF
					END_IF
				END_IF
			END_IF
			
			(* Valuta il Pass Mode Per L'asse Z *)
			IF Traiettoria^.PassModePoint_Z_Enable[1] THEN
				IF AsseZInMoto THEN
					IF Direzione_Z_Positiva THEN	//Se l'asse si sta muovendo in direzione POSITIVA
						IF ModuleAX_Z^.Ax^.Status.ActPosition >= (ProgrammaToModule_Z.Quota_Destinazione - OffsetPassMode.Z) THEN
							Asse_Z_InFinestraDiPassMode := TRUE;	
						END_IF
					ELSE							//Se l'asse si sta muovendo in direzione NEGATIVA
						IF ModuleAX_Z^.Ax^.Status.ActPosition <= (ProgrammaToModule_Z.Quota_Destinazione + OffsetPassMode.Z) THEN
							Asse_Z_InFinestraDiPassMode := TRUE;	
						END_IF
					END_IF
				END_IF
			END_IF
			
			(* Valuta il Pass Mode Per L'asse J *)
			IF Traiettoria^.PassModePoint_J_Enable[1] THEN
				IF AsseJInMoto THEN
					IF Direzione_J_Positiva THEN	//Se l'asse si sta muovendo in direzione POSITIVA
						IF ModuleAX_J^.Ax^.Status.ActPosition >= (ProgrammaToModule_J.Quota_Destinazione - OffsetPassMode.J) THEN
							Asse_J_InFinestraDiPassMode := TRUE;	
						END_IF
					ELSE							//Se l'asse si sta muovendo in direzione NEGATIVA
						IF ModuleAX_J^.Ax^.Status.ActPosition <= (ProgrammaToModule_J.Quota_Destinazione + OffsetPassMode.J) THEN
							Asse_J_InFinestraDiPassMode := TRUE;	
						END_IF
					END_IF
				END_IF
			END_IF
		(*
		WAMANAGER_CICLO_PRELIEVO_PACCO_RUN:
			(* Abilito tutti i pasmode*)
			Traiettoria^.PassModePoint_X_Enable[1] := TRUE; 
			Traiettoria^.PassModePoint_Y_Enable[1] := TRUE; 
			Traiettoria^.PassModePoint_Z_Enable[1] := TRUE;
			Traiettoria^.PassModePoint_J_Enable[1] := TRUE;
			Traiettoria^.PassModePoint_K_Enable[1] := TRUE;
			(* Valuta il Pass Mode Per L'asse X *)
			IF Traiettoria^.PassModePoint_X_Enable[1] THEN
				IF AsseXInMoto THEN
					IF Direzione_X_Positiva THEN	//Se l'asse si sta muovendo in direzione POSITIVA
						IF ModuleAX_X^.Ax^.Status.ActPosition >= (ProgrammaToModule_X.Quota_Destinazione - OffsetPassMode.X) THEN
							Asse_X_InFinestraDiPassMode := TRUE;	
						END_IF
					ELSE							//Se l'asse si sta muovendo in direzione NEGATIVA
						IF ModuleAX_X^.Ax^.Status.ActPosition <= (ProgrammaToModule_X.Quota_Destinazione + OffsetPassMode.X) THEN
							Asse_X_InFinestraDiPassMode := TRUE;	
						END_IF
					END_IF
				END_IF
			END_IF
				
			(* Valuta il Pass Mode Per L'asse Y *)
			IF Traiettoria^.PassModePoint_Y_Enable[1] THEN
				IF Pinza_InIngombroColonne_Attuale THEN
					OffsetPassModeY_Appoggio := 80;
				ELSE
					OffsetPassModeY_Appoggio := OffsetPassMode.Y;
				END_IF
				IF AsseYInMoto THEN
					IF Direzione_Y_Positiva THEN	//Se l'asse si sta muovendo in direzione POSITIVA
						IF ModuleAX_Y^.Ax^.Status.ActPosition >= (ProgrammaToModule_Y.Quota_Destinazione - OffsetPassModeY_Appoggio) THEN
							Asse_Y_InFinestraDiPassMode := TRUE;	
						END_IF
					ELSE							//Se l'asse si sta muovendo in direzione NEGATIVA
						IF ModuleAX_Y^.Ax^.Status.ActPosition <= (ProgrammaToModule_Y.Quota_Destinazione + OffsetPassModeY_Appoggio) THEN
							Asse_Y_InFinestraDiPassMode := TRUE;	
						END_IF
					END_IF
				END_IF
			END_IF
			
			(* Valuta il Pass Mode Per L'asse Z *)
			IF Traiettoria^.PassModePoint_Z_Enable[1] THEN
				IF AsseZInMoto THEN
					IF Direzione_Z_Positiva THEN	//Se l'asse si sta muovendo in direzione POSITIVA
						IF ModuleAX_Z^.Ax^.Status.ActPosition >= (ProgrammaToModule_Z.Quota_Destinazione - OffsetPassMode.Z) THEN
							Asse_Z_InFinestraDiPassMode := TRUE;	
						END_IF
					ELSE							//Se l'asse si sta muovendo in direzione NEGATIVA
						IF ModuleAX_Z^.Ax^.Status.ActPosition <= (ProgrammaToModule_Z.Quota_Destinazione + OffsetPassMode.Z) THEN
							Asse_Z_InFinestraDiPassMode := TRUE;	
						END_IF
					END_IF
				END_IF
			END_IF
			
			(* Valuta il Pass Mode Per L'asse J *)
			IF Traiettoria^.PassModePoint_J_Enable[1] THEN
				IF AsseJInMoto THEN
					IF Direzione_J_Positiva THEN	//Se l'asse si sta muovendo in direzione POSITIVA
						IF ModuleAX_J^.Ax^.Status.ActPosition >= (ProgrammaToModule_J.Quota_Destinazione - 2(*OffsetPassMode.J*)) THEN
							Asse_J_InFinestraDiPassMode := TRUE;	
						END_IF
					ELSE							//Se l'asse si sta muovendo in direzione NEGATIVA
						IF ModuleAX_J^.Ax^.Status.ActPosition <= (ProgrammaToModule_J.Quota_Destinazione + 2(*OffsetPassMode.J*)) THEN
							Asse_J_InFinestraDiPassMode := TRUE;	
						END_IF
					END_IF
				END_IF
			END_IF
									
		WAMANAGER_CICLO_DEPOSITO_PACCO_RUN:
			(* Abilito tutti i pasmode*)
			Traiettoria^.PassModePoint_X_Enable[1] := TRUE; 
			Traiettoria^.PassModePoint_Y_Enable[1] := TRUE; 
			Traiettoria^.PassModePoint_Z_Enable[1] := TRUE;
			Traiettoria^.PassModePoint_J_Enable[1] := TRUE;
			Traiettoria^.PassModePoint_K_Enable[1] := TRUE;
			(* Valuta il Pass Mode Per L'asse X *)
			IF Traiettoria^.PassModePoint_X_Enable[1] THEN
				IF AsseXInMoto THEN
					IF Direzione_X_Positiva THEN	//Se l'asse si sta muovendo in direzione POSITIVA
						IF ModuleAX_X^.Ax^.Status.ActPosition >= (ProgrammaToModule_X.Quota_Destinazione - OffsetPassMode.X) THEN
							Asse_X_InFinestraDiPassMode := TRUE;	
						END_IF
					ELSE							//Se l'asse si sta muovendo in direzione NEGATIVA
						IF ModuleAX_X^.Ax^.Status.ActPosition <= (ProgrammaToModule_X.Quota_Destinazione + OffsetPassMode.X) THEN
							Asse_X_InFinestraDiPassMode := TRUE;	
						END_IF
					END_IF
				END_IF
			END_IF
				
			(* Valuta il Pass Mode Per L'asse Y *)
			IF Traiettoria^.PassModePoint_Y_Enable[1] THEN
				IF AsseYInMoto THEN
					IF Direzione_Y_Positiva THEN	//Se l'asse si sta muovendo in direzione POSITIVA
						IF ModuleAX_Y^.Ax^.Status.ActPosition >= (ProgrammaToModule_Y.Quota_Destinazione - OffsetPassMode.Y) THEN
							Asse_Y_InFinestraDiPassMode := TRUE;	
						END_IF
					ELSE							//Se l'asse si sta muovendo in direzione NEGATIVA
						IF ModuleAX_Y^.Ax^.Status.ActPosition <= (ProgrammaToModule_Y.Quota_Destinazione + OffsetPassMode.Y) THEN
							Asse_Y_InFinestraDiPassMode := TRUE;	
						END_IF
					END_IF
				END_IF
			END_IF
			
			(* Valuta il Pass Mode Per L'asse Z *)
			IF Traiettoria^.PassModePoint_Z_Enable[1] THEN
				IF AsseZInMoto THEN
					IF Direzione_Z_Positiva THEN	//Se l'asse si sta muovendo in direzione POSITIVA
						IF ModuleAX_Z^.Ax^.Status.ActPosition >= (ProgrammaToModule_Z.Quota_Destinazione - OffsetPassMode.Z) THEN
							Asse_Z_InFinestraDiPassMode := TRUE;	
						END_IF
					ELSE							//Se l'asse si sta muovendo in direzione NEGATIVA
						IF ModuleAX_Z^.Ax^.Status.ActPosition <= (ProgrammaToModule_Z.Quota_Destinazione + OffsetPassMode.Z) THEN
							Asse_Z_InFinestraDiPassMode := TRUE;	
						END_IF
					END_IF
				END_IF
			END_IF
			
			(* Valuta il Pass Mode Per L'asse J *)
			IF Traiettoria^.PassModePoint_J_Enable[1] THEN
				IF AsseJInMoto THEN
					IF Direzione_J_Positiva THEN	//Se l'asse si sta muovendo in direzione POSITIVA
						IF ModuleAX_J^.Ax^.Status.ActPosition >= (ProgrammaToModule_J.Quota_Destinazione - OffsetPassMode.J) THEN
							Asse_J_InFinestraDiPassMode := TRUE;	
						END_IF
					ELSE							//Se l'asse si sta muovendo in direzione NEGATIVA
						IF ModuleAX_J^.Ax^.Status.ActPosition <= (ProgrammaToModule_J.Quota_Destinazione + OffsetPassMode.J) THEN
							Asse_J_InFinestraDiPassMode := TRUE;	
						END_IF
					END_IF
				END_IF
			END_IF
	*)
	END_CASE*)


ELSE
	(* Disabilito tutti i PasMode*)
	Traiettoria^.PassModePoint_X_Enable[1] := FALSE; 
	Traiettoria^.PassModePoint_Y_Enable[1] := FALSE; 
	Traiettoria^.PassModePoint_Z_Enable[1] := FALSE;
	Traiettoria^.PassModePoint_J_Enable[1] := FALSE;
	Traiettoria^.PassModePoint_K_Enable[1] := FALSE;
END_IF

END_FUNCTION_BLOCK

// ---- POUs/TFMachines/Utility/TFWorkflowsAllEnableOrDisable.TcPOU
//Funzione che restituisce TRUE se tutti i WORFLOW sono abilitati con ValutaEnable = TRUE o TRUE se tutti i WORFLOW sono disabilitati con ValutaEnable = FALSE
FUNCTION TFWorkflowsAllEnableOrDisable : BOOL 
VAR_INPUT
	WorkFlow : POINTER TO ARRAY[0..MAXWORKFLOW] OF WorkFlow;
	ValutaEnable : BOOL; // TRUE = Verifica se sono tutti enable, FALDE = se tutti disable
END_VAR
VAR
	i: UINT;
    nDisable : UINT;
	nEnable	: UINT;
END_VAR

FOR i:=0 TO MAXWORKFLOW DO
	IF WorkFlow^[i].Enable THEN
		nEnable := nEnable+1;
	ELSE
		nDisable := nDisable+1;
	END_IF
END_FOR
IF ValutaEnable THEN
	IF nEnable >= MAXWORKFLOW THEN
		TFWorkflowsAllEnableOrDisable := TRUE;
		RETURN;
	END_IF
ELSE
	IF nDisable >= MAXWORKFLOW THEN
		TFWorkflowsAllEnableOrDisable := TRUE;
		RETURN;
	END_IF
END_IF

END_FUNCTION

// ---- POUs/TFModules/Utility/TFPalletizerModulesCommandSend.TcPOU
FUNCTION TFPalletizerModulesCommandSend : BOOL (* Funzione che invia il comando a tutti i moduli della macchina *)
VAR_INPUT
	Cmd : UINT;
	ParametersArray : ParametersArray;
	Modules : POINTER TO TFPalletizerModules;
END_VAR
VAR
END_VAR

TFCommandSend(Cmd,ParametersArray,Modules^.AX_X.Cmd);
TFCommandSend(Cmd,ParametersArray,Modules^.AX_Y.Cmd);
TFCommandSend(Cmd,ParametersArray,Modules^.AX_Z.Cmd);
TFCommandSend(Cmd,ParametersArray,Modules^.AX_J.Cmd);
TFCommandSend(Cmd,ParametersArray,Modules^.Pinza.Cmd);

END_FUNCTION

// ---- POUs/TFModules/Utility/TFPalletizerModulesCheckState.TcPOU
FUNCTION TFPalletizerModulesCheckState : BOOL (* Funzione che ritorna TRUE se tutti i moduli sono nello stato richiesto *)
VAR_INPUT
	State : UINT;
	Modules : POINTER TO TFPalletizerModules;
END_VAR
VAR
END_VAR

TFPalletizerModulesCheckState	:=	
						TFStateCodeGet(Modules^.AX_X.State) = State AND
						TFStateCodeGet(Modules^.AX_Y.State) = State AND
						TFStateCodeGet(Modules^.AX_Z.State) = State AND 
						TFStateCodeGet(Modules^.AX_J.State) = State AND 
						TFStateCodeGet(Modules^.Pinza.State) = State;

END_FUNCTION

// ---- POUs/TFModules/Utility/TFPalletizerIsModuleError.TcPOU
//Funzione che ritorna TRUE se almeno un modulo è in errore
FUNCTION TFPalletizerIsModuleError : bool 
VAR_INPUT
	Modules : POINTER TO TFPalletizerModules;
END_VAR
VAR
END_VAR

TFPalletizerIsModuleError := TFIsModuleError(Modules^.AX_X.Error)OR
								TFIsModuleError(Modules^.AX_Y.Error)OR
								TFIsModuleError(Modules^.AX_Z.Error)OR
								TFIsModuleError(Modules^.AX_J.Error)OR
								TFIsModuleError(Modules^.Pinza.Error);

END_FUNCTION

// ---- POUs/TFModules/Utility/TFPalletizerModulesCheckPowerActive.TcPOU
FUNCTION TFPalletizerModulesCheckPowerActive : BOOL (* Funzione che ritorna TRUE se tutti gli assi sono in Power *)
VAR_INPUT
	Modules : POINTER TO TFPalletizerModules;
END_VAR
VAR
END_VAR

TFPalletizerModulesCheckPowerActive:=	
								 (Modules^.AX_X.Ax^.Status.PowerActive OR (Modules^.AX_X.Ax^.BrakeEnable AND Modules^.AX_X.Ax^.BrakePresent))AND
								 (Modules^.AX_Y.Ax^.Status.PowerActive OR (Modules^.AX_Y.Ax^.BrakeEnable AND Modules^.AX_Y.Ax^.BrakePresent))AND
								 (Modules^.AX_Z.Ax^.Status.PowerActive OR (Modules^.AX_Z.Ax^.BrakeEnable AND Modules^.AX_Z.Ax^.BrakePresent))AND
								 (Modules^.AX_J.Ax^.Status.PowerActive OR (Modules^.AX_J.Ax^.BrakeEnable AND Modules^.AX_J.Ax^.BrakePresent));

END_FUNCTION

// ---- POUs/TFMachines/Utility/TFIsWorkflowDisableOrEndedOrError.TcPOU
// Funzione che ritorna TRUE tutti i WORKFLOW sono almeno in uno dei seguenti stati: Disabilitato,Errore,Terminato
FUNCTION TFIsWorkflowDisableOrEndedOrError : BOOL 
VAR_INPUT
	NumWFPresence : UINT;
	WorkFlow : POINTER TO ARRAY[0..MAXWORKFLOW] OF WorkFlow;
END_VAR
VAR
	i: UINT;
END_VAR


FOR i:=0 TO NumWFPresence DO
	IF WorkFlow^[i].Enable = FALSE OR WorkFlow^[i].State = StateWF_END OR WorkFlow^[i].State = StateWF_END THEN
		TFIsWorkflowDisableOrEndedOrError := TRUE;
	ELSE
		TFIsWorkflowDisableOrEndedOrError := FALSE;
		RETURN;
	END_IF
END_FOR

END_FUNCTION

// ---- POUs/TFMachines/Utility/TFIsWorkflowError.TcPOU
// Funzione che ritorna TRUE se almeno un WORKFLOW è in errore
FUNCTION TFIsWorkflowError : BOOL 
VAR_INPUT
	WorkFlow : POINTER TO ARRAY[0..MAXWORKFLOW] OF WorkFlow;
END_VAR
VAR
	i: UINT;
END_VAR

FOR i:=0 TO MAXWORKFLOW DO
	IF WorkFlow^[i].State = StateWF_ERROR THEN
		TFIsWorkflowError := TRUE;
		RETURN;
	END_IF
END_FOR

END_FUNCTION

// ---- POUs/TFPalletizerDataTF/TFControlloInterferenza.TcPOU
FUNCTION TFControlloInterferenza : uINT
VAR_INPUT
	Traiettoria : POINTER TO TFTraiettoria;
	WorkSpace : POINTER TO TFMachinePalletizer_WorkSpace;
	WorkFootprint : POINTER TO ARRAY [1..MAXFOOTPRINT] OF TFMachinePalletizer_WorkFootprint;
	WorkPickPoint : POINTER TO ARRAY [1..MAXPICKPOINT] OF TFMachinePalletizer_WorkPickPointSlab;
	WorkArea : POINTER TO ARRAY [1..MAXAREA] OF TFMachinePalletizer_WorkArea;
	Pallet : POINTER TO ARRAY [1..MAXPALLET] OF TFMachinePalletizer_Pallet;
	Layer : POINTER TO ARRAY [1..MAXLAYER] OF TFMachinePalletizer_Layer;
	Forming : POINTER TO ARRAY [1..MAXFORMING] OF TFMachinePalletizer_FormingForSlab;
	
	Mission : POINTER TO TFMachinePalletizer_Mission;
	
	WorkAreaManager : POINTER TO TFWorkAreaManager;
	ModuleAX_X : POINTER TO TFModulePalletizer_Ax;
	ModuleAX_Y : POINTER TO TFModulePalletizer_Ax;
	ModuleAX_Z : POINTER TO TFModulePalletizer_Ax;
	ModuleAX_J : POINTER TO TFModulePalletizer_Ax;
	//ModuleAX_K : POINTER TO TFModulePalletizer_Ax;
END_VAR
VAR
	

END_VAR

TFControlloInterferenza := 0;

(* 1° Step - Check Start/End Points Inside WorkSpace *)
IF Traiettoria^.StartPoint.X < 0.0 OR Traiettoria^.StartPoint.X > WorkSpace^.X OR
	Traiettoria^.StartPoint.Y < 0.0 OR Traiettoria^.StartPoint.Y > WorkSpace^.Y OR
	Traiettoria^.StartPoint.Z < 0.0 OR Traiettoria^.StartPoint.Z > WorkSpace^.Z OR
	Traiettoria^.EndPoint.X < 0.0 OR Traiettoria^.EndPoint.X > WorkSpace^.X OR
	Traiettoria^.EndPoint.Y < 0.0 OR Traiettoria^.EndPoint.Y > WorkSpace^.Y OR
	(*Traiettoria^.EndPoint.Z < 0.0 OR*) Traiettoria^.EndPoint.Z > WorkSpace^.Z THEN
	TFControlloInterferenza := (ErrQUOTEDEPOSITO_NONCONFORMI); // Outside Limit
	RETURN;
END_IF

(* Controllo che le quote di fuori ingombro non superino il valore massimo ammesso dell'asse Z *)
IF QuotaFuoriIngombro_Z_ConFALDA >= WorkSpace^.Z AND (Mission^.State = MISSION_STATE_PRELIEVO_FALDA_RUN OR Mission^.State = MISSION_STATE_DEPOSITO_FALDA_RUN OR Mission^.State = MISSION_STATE_DEPOSITO_FALDA_DEPAL_RUN ) THEN
	TFControlloInterferenza := (ErrQUOTAZ_FALDAFUORIING_ELEVATA);
	RETURN;
ELSIF QuotaFuoriIngombro_Z_AVUOTO >= WorkSpace^.Z AND (Mission^.State <> MISSION_STATE_NOP) THEN
	TFControlloInterferenza := (ErrQUOTAZ_VUOTOFUORIING_ELEVATA);
	RETURN;
ELSIF QuotaFuoriIngombro_Z_ConPEZZO >= WorkSpace^.Z AND (Mission^.State = MISSION_STATE_PRELIEVO_LASTRA_DEPAL_RUN OR Mission^.State = MISSION_STATE_DEPOSITO_LASTRA_DEPAL_RUN) THEN
	TFControlloInterferenza := (ErrQUOTAZ_PACCOFUORIING_ELEVATA);
	RETURN;
END_IF

(* Controllo che gli assi abbiano quote "sensate" ovvero che rientrano nei limiti imposti dallo spazio di lavoro *)
IF ModuleAX_X^.Ax^.AxRef^.NcToPlc.ActPos >  ModuleAX_X^.Ax^.Parameter.MAXPosition OR 
	ModuleAX_X^.Ax^.AxRef^.NcToPlc.ActPos < ModuleAX_X^.Ax^.Parameter.MinPosition THEN
		TFControlloInterferenza := (ErroreACT_POSX_NONCONFORME);
		RETURN;
END_IF
IF ModuleAX_Y^.Ax^.AxRef^.NcToPlc.ActPos > ModuleAX_Y^.Ax^.Parameter.MAXPosition OR 
	ModuleAX_Y^.Ax^.AxRef^.NcToPlc.ActPos <  ModuleAX_Y^.Ax^.Parameter.MinPosition THEN
		TFControlloInterferenza := (ErroreACT_POSY_NONCONFORME);
		RETURN;
END_IF
IF ModuleAX_Z^.Ax^.AxRef^.NcToPlc.ActPos > ModuleAX_Z^.Ax^.Parameter.MAXPosition OR 
	ModuleAX_Z^.Ax^.AxRef^.NcToPlc.ActPos <  ModuleAX_Z^.Ax^.Parameter.MinPosition THEN 
		TFControlloInterferenza := (ErroreACT_POSZ_NONCONFORME);
		RETURN;
END_IF
IF ModuleAX_J^.Ax^.AxRef^.NcToPlc.ActPos > ModuleAX_J^.Ax^.Parameter.MAXPosition OR 
	ModuleAX_J^.Ax^.AxRef^.NcToPlc.ActPos <  ModuleAX_J^.Ax^.Parameter.MinPosition THEN 
		TFControlloInterferenza := (ErroreACT_POSJ_NONCONFORME);
		RETURN;
END_IF

END_FUNCTION

// ---- POUs/TFPalletizerDataTF/TFCalcoloVelocita.TcPOU
FUNCTION TFCalcoloVelocita : BOOL
VAR_INPUT
	AxisOverride : POINTER TO TFMachinePalletizer_VelocityOverride_TF;
	Mission : POINTER TO TFMachinePalletizer_Mission;
	ArrayPacchi : POINTER TO DUT_ArrayPacchi; 					//Array contenente i pacchi sui trasporti				
	DepositoPaccoInLenta : BOOL;
END_VAR
VAR
	NUltimiTrasportiOccupati : UINT;
	OverrideAutomatico	: REAL;
	OverrideCicloPallet	: REAL;
	OverrideCicloPacco	: REAL;
	OverrideCicloFalda	: REAL;
	OverrideCicloJog	: REAL;
	OverrideCicloRiposo	: REAL;
	
	OverrideGlobaleCicloPallet  : REAL; 	
	OverrideGlobaleCicloPacco 	: REAL;	
	OverrideGlobaleCicloFalda 	: REAL; 	
	OverrideGlobaleCicloJog 	: REAL;
	OverrideGlobaleCicloAvuoto	: REAL;
	
	OverrideAutomaticoOLD: REAL;
END_VAR

TFCalcoloVelocita := FALSE;

(* Trasferimento valori da variabile scritta da HMI a variabile Globale *)

AxisOverride^.Auto := HMI_AxisOverride.Auto;
AxisOverride^.Jog := HMI_AxisOverride.Jog;
AxisOverride^.Layer := HMI_AxisOverride.Layer;
IF Mission^.XDim >= 3100 THEN//se formato maggiore di 2900 seghiamo override al 80%
	HMI_AxisOverride.Pack := MIN(80,HMI_AxisOverride.Pack);
END_IF
AxisOverride^.Pack := HMI_AxisOverride.Pack;
AxisOverride^.Pallet := HMI_AxisOverride.Pallet;
AxisOverride^.Riposo := HMI_AxisOverride.PickRip;

IF FROM_HMI_PAL.HMI_AbilitaOverrideDinamico AND FALSE THEN
	NUltimiTrasportiOccupati := TFNumeroUltimi_N_TrasportiOccupati(ArrayPacchi,7);;//TFNumeroUltimi_N_TrasportiOccupati(HandlingPackTable,7);
	OverrideAutomatico := (AxisOverride^.Auto/100) * (TFCalcoloOverrideDinamico(NUltimiTrasportiOccupati,HMI_OverideDinamico)/100);
	IF NUltimiTrasportiOccupati > 0 THEN
		OverrideAutomaticoOLD := OverrideAutomatico;
	END_IF
	IF OverrideAutomatico = 0 THEN
		IF OverrideAutomaticoOLD <= 0 THEN
			OverrideAutomatico 	:= AxisOverride^.Auto/100;
		ELSE
			OverrideAutomatico := OverrideAutomaticoOLD;
		END_IF
	END_IF
ELSE
	OverrideAutomatico 	:= AxisOverride^.Auto/100;	
END_IF

IF OverrideAutomatico <= 0.01 THEN
	OverrideAutomatico := 1;
END_IF

//OverrideAutomatico 	:= AxisOverride^.Auto/ 100;	
OverrideCicloPallet := AxisOverride^.Pallet/ 100;	
OverrideCicloPacco 	:= AxisOverride^.Pack/ 100;	
OverrideCicloFalda 	:= AxisOverride^.Layer/ 100;	
OverrideCicloJog 	:= AxisOverride^.Jog/ 100;	
OverrideCicloRiposo	:= AxisOverride^.Riposo/ 100;	

OverrideGlobaleCicloPallet  := OverrideAutomatico * OverrideCicloPallet;  	
OverrideGlobaleCicloPacco 	:= OverrideAutomatico *	OverrideCicloPacco;
OverrideGlobaleCicloFalda 	:= OverrideAutomatico *	OverrideCicloFalda;
OverrideGlobaleCicloJog 	:= OverrideAutomatico * OverrideCicloJog;
OverrideGlobaleCicloAvuoto 	:= OverrideAutomatico * OverrideCicloRiposo;


HMI_ParametriAsseX_CicloFalda.Vel_Ridotta 	:= MIN(HMI_ParametriAsseX_CicloFalda.Vel_Ridotta,10);
HMI_ParametriAsseX_CicloPacco.Vel_Ridotta 	:= MIN(HMI_ParametriAsseX_CicloPacco.Vel_Ridotta,10);
HMI_ParametriAsseX_CicloPallet.Vel_Ridotta 	:= MIN(HMI_ParametriAsseX_CicloPallet.Vel_Ridotta,10);
HMI_ParametriAsseX_CicloRiposo.Vel_Ridotta 	:= MIN(HMI_ParametriAsseX_CicloRiposo.Vel_Ridotta,10);

HMI_ParametriAsseY_CicloFalda.Vel_Ridotta 	:= MIN(HMI_ParametriAsseY_CicloFalda.Vel_Ridotta,2);
HMI_ParametriAsseY_CicloPacco.Vel_Ridotta 	:= MIN(HMI_ParametriAsseY_CicloPacco.Vel_Ridotta,2);
HMI_ParametriAsseY_CicloPallet.Vel_Ridotta 	:= MIN(HMI_ParametriAsseY_CicloPallet.Vel_Ridotta,2);
HMI_ParametriAsseY_CicloRiposo.Vel_Ridotta 	:= MIN(HMI_ParametriAsseY_CicloRiposo.Vel_Ridotta,2);

HMI_ParametriAsseZ_CicloFalda.Vel_Ridotta 	:= MIN(HMI_ParametriAsseZ_CicloFalda.Vel_Ridotta,10);
HMI_ParametriAsseZ_CicloPacco.Vel_Ridotta 	:= MIN(HMI_ParametriAsseZ_CicloPacco.Vel_Ridotta,10);
HMI_ParametriAsseZ_CicloPallet.Vel_Ridotta 	:= MIN(HMI_ParametriAsseZ_CicloPallet.Vel_Ridotta,10);
HMI_ParametriAsseZ_CicloRiposo.Vel_Ridotta 	:= MIN(HMI_ParametriAsseZ_CicloRiposo.Vel_Ridotta,10);

HMI_ParametriAsseJ_CicloFalda.Vel_Ridotta 	:= MIN(HMI_ParametriAsseJ_CicloFalda.Vel_Ridotta,10);
HMI_ParametriAsseJ_CicloPacco.Vel_Ridotta 	:= MIN(HMI_ParametriAsseJ_CicloPacco.Vel_Ridotta,10);
HMI_ParametriAsseJ_CicloPallet.Vel_Ridotta 	:= MIN(HMI_ParametriAsseJ_CicloPallet.Vel_Ridotta,10);
HMI_ParametriAsseJ_CicloRiposo.Vel_Ridotta 	:= MIN(HMI_ParametriAsseJ_CicloRiposo.Vel_Ridotta,10);


////////////////////////////////////////////////////////////////////////////////////////////////////////////////////////////////////////////////
//////////////////////////////////////////////////// CICLO DI RIPOSO ///////////////////////////////////////////////////////////////////////////
////////////////////////////////////////////////////////////////////////////////////////////////////////////////////////////////////////////////

	HMI_ParametriAsseX_CicloRiposo.Acc_Carico	:= MAX(1,HMI_ParametriAsseX_CicloRiposo.Acc_Carico);
	HMI_ParametriAsseX_CicloRiposo.Acc_Vuoto	:= MAX(1,HMI_ParametriAsseX_CicloRiposo.Acc_Vuoto); 
																						
	HMI_ParametriAsseY_CicloRiposo.Acc_Carico	:= MAX(1,HMI_ParametriAsseY_CicloRiposo.Acc_Carico);
	HMI_ParametriAsseY_CicloRiposo.Acc_Vuoto	:= MAX(1,HMI_ParametriAsseY_CicloRiposo.Acc_Vuoto); 
																						
	HMI_ParametriAsseZ_CicloRiposo.Acc_Carico	:= MAX(1,HMI_ParametriAsseZ_CicloRiposo.Acc_Carico);
	HMI_ParametriAsseZ_CicloRiposo.Acc_Vuoto	:= MAX(1,HMI_ParametriAsseZ_CicloRiposo.Acc_Vuoto); 
																						
	HMI_ParametriAsseJ_CicloRiposo.Acc_Carico	:= MAX(1,HMI_ParametriAsseJ_CicloRiposo.Acc_Carico);
	HMI_ParametriAsseJ_CicloRiposo.Acc_Vuoto	:= MAX(1,HMI_ParametriAsseJ_CicloRiposo.Acc_Vuoto); 
																					   
	HMI_ParametriAsseK_CicloRiposo.Acc_Carico	:= MAX(1,HMI_ParametriAsseK_CicloRiposo.Acc_Carico);
	HMI_ParametriAsseK_CicloRiposo.Acc_Vuoto	:= MAX(1,HMI_ParametriAsseK_CicloRiposo.Acc_Vuoto); 

	HMI_ParametriAsseX_CicloRiposo.Vel_Carico	:= MAX(1,HMI_ParametriAsseX_CicloRiposo.Vel_Carico);	
	HMI_ParametriAsseX_CicloRiposo.Vel_Ridotta  := MAX(1,HMI_ParametriAsseX_CicloRiposo.Vel_Ridotta);
		

	HMI_ParametriAsseX_CicloRiposo.Dec_Carico 		:= HMI_ParametriAsseX_CicloRiposo.Acc_Carico;
	HMI_ParametriAsseX_CicloRiposo.Dec_Vuoto  		:= HMI_ParametriAsseX_CicloRiposo.Acc_Vuoto;

	HMI_ParametriAsseY_CicloRiposo.Dec_Carico 		:= HMI_ParametriAsseY_CicloRiposo.Acc_Carico;
	HMI_ParametriAsseY_CicloRiposo.Dec_Vuoto  		:= HMI_ParametriAsseY_CicloRiposo.Acc_Vuoto;
		
	HMI_ParametriAsseZ_CicloRiposo.Dec_Carico 		:= HMI_ParametriAsseZ_CicloRiposo.Acc_Carico;
	HMI_ParametriAsseZ_CicloRiposo.Dec_Vuoto  		:= HMI_ParametriAsseZ_CicloRiposo.Acc_Vuoto;
	
	HMI_ParametriAsseJ_CicloRiposo.Dec_Carico 		:= HMI_ParametriAsseJ_CicloRiposo.Acc_Carico;
	HMI_ParametriAsseJ_CicloRiposo.Dec_Vuoto  		:= HMI_ParametriAsseJ_CicloRiposo.Acc_Vuoto;
	
	HMI_ParametriAsseK_CicloRiposo.Dec_Carico 		:= HMI_ParametriAsseK_CicloRiposo.Acc_Carico;
	HMI_ParametriAsseK_CicloRiposo.Dec_Vuoto  		:= HMI_ParametriAsseK_CicloRiposo.Acc_Vuoto;
	
	(* ASSE X *)
	
	ParametriProgramma_X_CicloRiposo.Acc_Carico		:= AxisNominalPar_X.MaximumAcceleration * (HMI_ParametriAsseX_CicloRiposo.Acc_Carico/100);
	ParametriProgramma_X_CicloRiposo.Acc_Vuoto		:= AxisNominalPar_X.MaximumAcceleration * (HMI_ParametriAsseX_CicloRiposo.Acc_Vuoto/100);
	ParametriProgramma_X_CicloRiposo.Dec_Carico 	:= AxisNominalPar_X.MaximumDeceleration * (HMI_ParametriAsseX_CicloRiposo.Dec_Carico/100);
	ParametriProgramma_X_CicloRiposo.Dec_Vuoto  	:= AxisNominalPar_X.MaximumDeceleration * (HMI_ParametriAsseX_CicloRiposo.Dec_Vuoto/100);
	ParametriProgramma_X_CicloRiposo.Jerk_Carico  	:= AxisNominalPar_X.DefaultJerk * 		  (HMI_ParametriAsseX_CicloRiposo.Jerk_Carico/100);
	ParametriProgramma_X_CicloRiposo.Jerk_Vuoto  	:= AxisNominalPar_X.DefaultJerk * 		  (HMI_ParametriAsseX_CicloRiposo.Jerk_Vuoto/100);
	ParametriProgramma_X_CicloRiposo.Torque  		:= AxisNominalPar_X.DefaultTorque * 	  (HMI_ParametriAsseX_CicloRiposo.Torque/100);
	ParametriProgramma_X_CicloRiposo.Vel_Carico  	:= AxisNominalPar_X.ReferenceVelocity *   (HMI_ParametriAsseX_CicloRiposo.Vel_Carico/100) * OverrideGlobaleCicloAvuoto;
	ParametriProgramma_X_CicloRiposo.Vel_Ridotta  	:= AxisNominalPar_X.ReferenceVelocity *   (HMI_ParametriAsseX_CicloRiposo.Vel_Ridotta/100);// * OverrideGlobaleCicloAvuoto;
	ParametriProgramma_X_CicloRiposo.Vel_Vuoto  	:= AxisNominalPar_X.ReferenceVelocity *   (HMI_ParametriAsseX_CicloRiposo.Vel_Vuoto/100) * OverrideGlobaleCicloAvuoto;
	
	(* ASSE Y *)
		
	ParametriProgramma_Y_CicloRiposo.Acc_Carico		:= AxisNominalPar_Y.MaximumAcceleration * (HMI_ParametriAsseY_CicloRiposo.Acc_Carico/100);
	ParametriProgramma_Y_CicloRiposo.Acc_Vuoto		:= AxisNominalPar_Y.MaximumAcceleration * (HMI_ParametriAsseY_CicloRiposo.Acc_Vuoto/100);
	ParametriProgramma_Y_CicloRiposo.Dec_Carico 	:= AxisNominalPar_Y.MaximumDeceleration * (HMI_ParametriAsseY_CicloRiposo.Dec_Carico/100);
	ParametriProgramma_Y_CicloRiposo.Dec_Vuoto  	:= AxisNominalPar_Y.MaximumDeceleration * (HMI_ParametriAsseY_CicloRiposo.Dec_Vuoto/100);
	ParametriProgramma_Y_CicloRiposo.Jerk_Carico  	:= AxisNominalPar_Y.DefaultJerk * (HMI_ParametriAsseY_CicloRiposo.Jerk_Carico/100);
	ParametriProgramma_Y_CicloRiposo.Jerk_Vuoto  	:= AxisNominalPar_Y.DefaultJerk * (HMI_ParametriAsseY_CicloRiposo.Jerk_Vuoto/100);
	ParametriProgramma_Y_CicloRiposo.Torque  		:= AxisNominalPar_Y.DefaultTorque * (HMI_ParametriAsseY_CicloRiposo.Torque/100);
	ParametriProgramma_Y_CicloRiposo.Vel_Carico  	:= AxisNominalPar_Y.ReferenceVelocity * (HMI_ParametriAsseY_CicloRiposo.Vel_Carico/100) * OverrideGlobaleCicloAvuoto;
	ParametriProgramma_Y_CicloRiposo.Vel_Ridotta  	:= AxisNominalPar_Y.ReferenceVelocity * (HMI_ParametriAsseY_CicloRiposo.Vel_Ridotta/100);// * OverrideGlobaleCicloAvuoto;
	ParametriProgramma_Y_CicloRiposo.Vel_Vuoto  	:= AxisNominalPar_Y.ReferenceVelocity * (HMI_ParametriAsseY_CicloRiposo.Vel_Vuoto/100) * OverrideGlobaleCicloAvuoto;
	
	(* ASSE Z *)
		
	ParametriProgramma_Z_CicloRiposo.Acc_Carico		:= AxisNominalPar_Z.MaximumAcceleration * (HMI_ParametriAsseZ_CicloRiposo.Acc_Carico/100);
	ParametriProgramma_Z_CicloRiposo.Acc_Vuoto		:= AxisNominalPar_Z.MaximumAcceleration * (HMI_ParametriAsseZ_CicloRiposo.Acc_Vuoto/100);
	ParametriProgramma_Z_CicloRiposo.Dec_Carico 	:= AxisNominalPar_Z.MaximumDeceleration * (HMI_ParametriAsseZ_CicloRiposo.Dec_Carico/100);
	ParametriProgramma_Z_CicloRiposo.Dec_Vuoto  	:= AxisNominalPar_Z.MaximumDeceleration * (HMI_ParametriAsseZ_CicloRiposo.Dec_Vuoto/100);
	ParametriProgramma_Z_CicloRiposo.Jerk_Carico  	:= AxisNominalPar_Z.DefaultJerk * (HMI_ParametriAsseZ_CicloRiposo.Jerk_Carico/100);
	ParametriProgramma_Z_CicloRiposo.Jerk_Vuoto  	:= AxisNominalPar_Z.DefaultJerk * (HMI_ParametriAsseZ_CicloRiposo.Jerk_Vuoto/100);
	ParametriProgramma_Z_CicloRiposo.Torque  		:= AxisNominalPar_Z.DefaultTorque * (HMI_ParametriAsseZ_CicloRiposo.Torque/100);
	ParametriProgramma_Z_CicloRiposo.Vel_Carico  	:= AxisNominalPar_Z.ReferenceVelocity * (HMI_ParametriAsseZ_CicloRiposo.Vel_Carico/100) * OverrideGlobaleCicloAvuoto;
	ParametriProgramma_Z_CicloRiposo.Vel_Ridotta  	:= AxisNominalPar_Z.ReferenceVelocity * (HMI_ParametriAsseZ_CicloRiposo.Vel_Ridotta/100);// * OverrideGlobaleCicloRiposo;
	ParametriProgramma_Z_CicloRiposo.Vel_Vuoto  	:= AxisNominalPar_Z.ReferenceVelocity * (HMI_ParametriAsseZ_CicloRiposo.Vel_Vuoto/100) * OverrideGlobaleCicloAvuoto;
	
	(* ASSE J *)
	
	ParametriProgramma_J_CicloRiposo.Acc_Carico		:= AxisNominalPar_J.MaximumAcceleration * (HMI_ParametriAsseJ_CicloRiposo.Acc_Carico/100);
	ParametriProgramma_J_CicloRiposo.Acc_Vuoto		:= AxisNominalPar_J.MaximumAcceleration * (HMI_ParametriAsseJ_CicloRiposo.Acc_Vuoto/100);
	ParametriProgramma_J_CicloRiposo.Dec_Carico 	:= AxisNominalPar_J.MaximumDeceleration * (HMI_ParametriAsseJ_CicloRiposo.Dec_Carico/100);
	ParametriProgramma_J_CicloRiposo.Dec_Vuoto  	:= AxisNominalPar_J.MaximumDeceleration * (HMI_ParametriAsseJ_CicloRiposo.Dec_Vuoto/100);
	ParametriProgramma_J_CicloRiposo.Jerk_Carico  	:= AxisNominalPar_J.DefaultJerk * (HMI_ParametriAsseJ_CicloRiposo.Jerk_Carico/100);
	ParametriProgramma_J_CicloRiposo.Jerk_Vuoto  	:= AxisNominalPar_J.DefaultJerk * (HMI_ParametriAsseJ_CicloRiposo.Jerk_Vuoto/100);
	ParametriProgramma_J_CicloRiposo.Torque  		:= AxisNominalPar_J.DefaultTorque * (HMI_ParametriAsseJ_CicloRiposo.Torque/100);
	ParametriProgramma_J_CicloRiposo.Vel_Carico  	:= AxisNominalPar_J.ReferenceVelocity * (HMI_ParametriAsseJ_CicloRiposo.Vel_Carico/100);// * OverrideGlobaleCicloAvuoto;
	ParametriProgramma_J_CicloRiposo.Vel_Ridotta  	:= AxisNominalPar_J.ReferenceVelocity * (HMI_ParametriAsseJ_CicloRiposo.Vel_Ridotta/100);// * OverrideGlobaleCicloAvuoto;
	ParametriProgramma_J_CicloRiposo.Vel_Vuoto  	:= AxisNominalPar_J.ReferenceVelocity * (HMI_ParametriAsseJ_CicloRiposo.Vel_Vuoto/100);// * OverrideGlobaleCicloAvuoto;
	(* ASSE K *)
	(*
	ParametriProgramma_K_CicloRiposo.Acc_Carico		:= AxisNominalPar_K.MaximumAcceleration * (HMI_ParametriAsseK_CicloRiposo.Acc_Carico/100);
	ParametriProgramma_K_CicloRiposo.Acc_Vuoto		:= AxisNominalPar_K.MaximumAcceleration * (HMI_ParametriAsseK_CicloRiposo.Acc_Vuoto/100);
	ParametriProgramma_K_CicloRiposo.Dec_Carico 	:= AxisNominalPar_K.MaximumDeceleration * (HMI_ParametriAsseK_CicloRiposo.Dec_Carico/100);
	ParametriProgramma_K_CicloRiposo.Dec_Vuoto  	:= AxisNominalPar_K.MaximumDeceleration * (HMI_ParametriAsseK_CicloRiposo.Dec_Vuoto/100);
	ParametriProgramma_K_CicloRiposo.Jerk_Carico  	:= AxisNominalPar_K.DefaultJerk * (HMI_ParametriAsseK_CicloRiposo.Jerk_Carico/100);
	ParametriProgramma_K_CicloRiposo.Jerk_Vuoto  	:= AxisNominalPar_K.DefaultJerk * (HMI_ParametriAsseK_CicloRiposo.Jerk_Vuoto/100);
	//ParametriProgramma_K_CicloRiposo.Torque  		:= Mission^.KPickTorque;//AxisNominalPar_K.DefaultTorque * (HMI_ParametriAsseK_CicloRiposo.Torque/100);
	ParametriProgramma_K_CicloRiposo.Vel_Carico  	:= AxisNominalPar_K.ReferenceVelocity * (HMI_ParametriAsseK_CicloRiposo.Vel_Carico/100);// * OverrideGlobaleCicloAvuoto;
	ParametriProgramma_K_CicloRiposo.Vel_Ridotta  	:= AxisNominalPar_K.ReferenceVelocity * (HMI_ParametriAsseK_CicloRiposo.Vel_Ridotta/100);// * OverrideGlobaleCicloAvuoto;
	ParametriProgramma_K_CicloRiposo.Vel_Vuoto  	:= AxisNominalPar_K.ReferenceVelocity * (HMI_ParametriAsseK_CicloRiposo.Vel_Vuoto/100);//* OverrideGlobaleCicloAvuoto;
	*)
////////////////////////////////////////////////////////////////////////////////////////////////////////////////////////////////////////////////
//////////////////////////////////////////////////// CICLO FALDA //////////////////////////////////////////////////////////////////////////////
////////////////////////////////////////////////////////////////////////////////////////////////////////////////////////////////////////////////

	HMI_ParametriAsseX_CicloFalda.Acc_Carico	:= MAX(1,HMI_ParametriAsseX_CicloFalda.Acc_Carico);
	HMI_ParametriAsseX_CicloFalda.Acc_Vuoto		:= MAX(1,HMI_ParametriAsseX_CicloFalda.Acc_Vuoto); 
																				 
	HMI_ParametriAsseY_CicloFalda.Acc_Carico	:= MAX(1,HMI_ParametriAsseY_CicloFalda.Acc_Carico);
	HMI_ParametriAsseY_CicloFalda.Acc_Vuoto		:= MAX(1,HMI_ParametriAsseY_CicloFalda.Acc_Vuoto); 
																				 
	HMI_ParametriAsseZ_CicloFalda.Acc_Carico	:= MAX(1,HMI_ParametriAsseZ_CicloFalda.Acc_Carico);
	HMI_ParametriAsseZ_CicloFalda.Acc_Vuoto		:= MAX(1,HMI_ParametriAsseZ_CicloFalda.Acc_Vuoto); 
																				 
	HMI_ParametriAsseJ_CicloFalda.Acc_Carico	:= MAX(1,HMI_ParametriAsseJ_CicloFalda.Acc_Carico);
	HMI_ParametriAsseJ_CicloFalda.Acc_Vuoto		:= MAX(1,HMI_ParametriAsseJ_CicloFalda.Acc_Vuoto); 
																			     
	HMI_ParametriAsseK_CicloFalda.Acc_Carico	:= MAX(1,HMI_ParametriAsseK_CicloFalda.Acc_Carico);
	HMI_ParametriAsseK_CicloFalda.Acc_Vuoto		:= MAX(1,HMI_ParametriAsseK_CicloFalda.Acc_Vuoto); 
                                                                                 
	HMI_ParametriAsseX_CicloFalda.Vel_Carico	:= MAX(1,HMI_ParametriAsseX_CicloFalda.Vel_Carico);	
	HMI_ParametriAsseX_CicloFalda.Vel_Ridotta  	:= MAX(1,HMI_ParametriAsseX_CicloFalda.Vel_Ridotta);
	

	HMI_ParametriAsseX_CicloFalda.Dec_Carico 		:= HMI_ParametriAsseX_CicloFalda.Acc_Carico;
	HMI_ParametriAsseX_CicloFalda.Dec_Vuoto  		:= HMI_ParametriAsseX_CicloFalda.Acc_Vuoto;

	HMI_ParametriAsseY_CicloFalda.Dec_Carico 		:= HMI_ParametriAsseY_CicloFalda.Acc_Carico;
	HMI_ParametriAsseY_CicloFalda.Dec_Vuoto  		:= HMI_ParametriAsseY_CicloFalda.Acc_Vuoto;
		
	HMI_ParametriAsseZ_CicloFalda.Dec_Carico 		:= HMI_ParametriAsseZ_CicloFalda.Acc_Carico;
	HMI_ParametriAsseZ_CicloFalda.Dec_Vuoto  		:= HMI_ParametriAsseZ_CicloFalda.Acc_Vuoto;
	
